KUKA KRL program: f1_Kuka_APT215T02S15.SRC

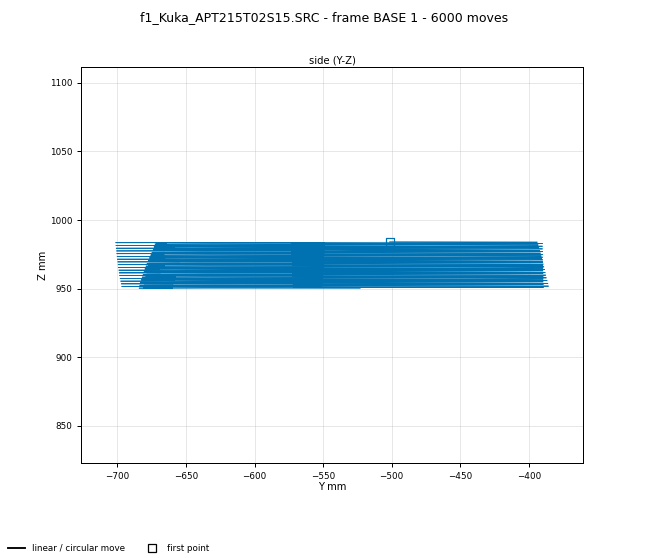
[picture p0: tool path of f1_Kuka_APT215T02S15.SRC in frame BASE 1, 6000 of 6001 moves have a stored position in this frame; points joined in program order, loops and branches not executed]
&ACCESS RVP
&REL 2
&PARAM TEMPLATE = C:\KRC\Roboter\Template\vorgabe
&PARAM EDITMASK = *
DEF f1_Kuka_APT215T02S15()


;FOLD INI;%{PE}%V3.2.0,%MKUKATPBASIS,%CINIT,%VCOMMON,%P
  ;FOLD BAS INI;%{E}%V3.2.0,%MKUKATPBASIS,%CINIT,%VINIT,%P
    GLOBAL INTERRUPT DECL 3 WHEN $STOPMESS==TRUE DO IR_STOPM ( )
    INTERRUPT ON 3
    BAS (#INITMOV,0 )
  ;ENDFOLD (BAS INI)
  ;FOLD USER INI;%{E}%V3.2.0,%MKUKATPUSER,%CINIT,%VINIT,%P
    ;Make your modifications here
  ;ENDFOLD (USER INI)
;ENDFOLD (INI)


;*** Make Null PTP Move
  PTP $pos_act

;*** Auto Load The Correct TOOL Data
  $tool=tool_data[2]

;*** Auto Load The Correct BASE Data
  $base=base_data[1]

  $ADVANCE = 5

;*** Restate Last Velocity
MMPM(30000.0)
SetRPM(8000)
LIN {X -0.285,Y -501.480,Z 984.115,A 0.000,B 0.000,C 90.000,E1 236.707} C_DIS
LIN {X 0.055,Y -498.844,Z 984.108,A 0.000,B 0.000,C 90.000,E1 235.468} C_DIS
LIN {X 0.071,Y -494.695,Z 984.098,A 0.000,B 0.000,C 90.000,E1 233.657} C_DIS
LIN {X -0.059,Y -492.503,Z 984.093,A 0.000,B 0.000,C 90.000,E1 232.763} C_DIS
LIN {X 0.019,Y -488.185,Z 984.083,A 0.000,B 0.000,C 90.000,E1 230.928} C_DIS
LIN {X 0.171,Y -484.612,Z 984.075,A 0.000,B 0.000,C 90.000,E1 229.380} C_DIS
LIN {X 0.130,Y -479.643,Z 984.063,A 0.000,B 0.000,C 90.000,E1 227.229} C_DIS
LIN {X -0.171,Y -475.684,Z 984.052,A 0.000,B 0.000,C 90.000,E1 225.405} C_DIS
LIN {X 0.017,Y -472.371,Z 984.044,A 0.000,B 0.000,C 90.000,E1 223.824} C_DIS
LIN {X 0.143,Y -468.887,Z 984.035,A 0.000,B 0.000,C 90.000,E1 222.243} C_DIS
LIN {X -0.119,Y -465.376,Z 984.026,A 0.000,B 0.000,C 90.000,E1 220.701} C_DIS
LIN {X 0.008,Y -461.153,Z 984.016,A 0.000,B 0.000,C 90.000,E1 218.785} C_DIS
LIN {X -0.234,Y -456.180,Z 984.003,A 0.000,B 0.000,C 90.000,E1 216.583} C_DIS
LIN {X 0.053,Y -453.348,Z 983.996,A 0.000,B 0.000,C 90.000,E1 215.264} C_DIS
LIN {X -0.282,Y -449.138,Z 983.985,A 0.000,B 0.000,C 90.000,E1 213.372} C_DIS
LIN {X -0.043,Y -445.627,Z 983.976,A 0.000,B 0.000,C 90.000,E1 211.720} C_DIS
LIN {X 0.037,Y -442.148,Z 983.967,A 0.000,B 0.000,C 90.000,E1 210.079} C_DIS
LIN {X 0.229,Y -439.200,Z 983.960,A 0.000,B 0.000,C 90.000,E1 208.743} C_DIS
LIN {X 0.220,Y -433.424,Z 983.945,A 0.000,B 0.000,C 90.000,E1 206.104} C_DIS
LIN {X -0.144,Y -430.325,Z 983.938,A 0.000,B 0.000,C 90.000,E1 204.823} C_DIS
LIN {X 0.213,Y -425.721,Z 983.927,A 0.000,B 0.000,C 90.000,E1 202.770} C_DIS
LIN {X 0.085,Y -420.612,Z 983.914,A 0.000,B 0.000,C 90.000,E1 200.429} C_DIS
LIN {X 0.213,Y -414.989,Z 983.898,A 0.000,B 0.000,C 90.000,E1 197.692} C_DIS
LIN {X 0.183,Y -409.982,Z 983.883,A 0.000,B 0.000,C 90.000,E1 194.954} C_DIS
LIN {X 0.056,Y -407.467,Z 983.876,A 0.000,B 0.000,C 90.000,E1 193.592} C_DIS
LIN {X -0.202,Y -405.003,Z 983.868,A 0.000,B 0.000,C 90.000,E1 192.243} C_DIS
LIN {X -0.103,Y -401.708,Z 983.858,A 0.000,B 0.000,C 90.000,E1 190.489} C_DIS
LIN {X -0.128,Y -399.174,Z 983.850,A 0.000,B 0.000,C 90.000,E1 189.095} C_DIS
LIN {X 0.168,Y -396.164,Z 983.841,A 0.000,B 0.000,C 90.000,E1 187.296} C_DIS
LIN {X 0.061,Y -395.147,Z 983.837,A 0.000,B 0.000,C 90.000,E1 186.606} C_DIS
LIN {X -0.088,Y -394.070,Z 983.831,A 0.000,B 0.000,C 90.000,E1 185.568} C_DIS
LIN {X -0.208,Y -393.751,Z 983.827,A 0.000,B 0.000,C 90.000,E1 184.878} C_DIS
LIN {X 0.062,Y -393.914,Z 983.823,A 0.000,B 0.000,C 90.000,E1 184.131} C_DIS
LIN {X -0.062,Y -394.851,Z 983.819,A 0.000,B 0.000,C 90.000,E1 183.440} C_DIS
LIN {X -0.092,Y -396.130,Z 983.816,A 0.000,B 0.000,C 90.000,E1 182.922} C_DIS
LIN {X -0.126,Y -399.219,Z 983.812,A 0.000,B 0.000,C 90.000,E1 182.178} C_DIS
LIN {X -0.178,Y -401.986,Z 983.809,A 0.000,B 0.000,C 90.000,E1 181.718} C_DIS
LIN {X -0.127,Y -405.589,Z 983.807,A 0.000,B 0.000,C 90.000,E1 181.203} C_DIS
LIN {X -0.089,Y -413.849,Z 983.802,A 0.000,B 0.000,C 90.000,E1 180.286} C_DIS
LIN {X -0.065,Y -430.114,Z 983.793,A 0.000,B 0.000,C 90.000,E1 178.682} C_DIS
LIN {X -0.102,Y -437.269,Z 983.789,A 0.000,B 0.000,C 90.000,E1 177.993} C_DIS
LIN {X -0.024,Y -444.519,Z 983.785,A 0.000,B 0.000,C 90.000,E1 177.249} C_DIS
LIN {X -0.047,Y -454.485,Z 983.779,A 0.000,B 0.000,C 90.000,E1 176.216} C_DIS
LIN {X -0.161,Y -462.529,Z 983.774,A 0.000,B 0.000,C 90.000,E1 175.355} C_DIS
LIN {X -0.135,Y -470.477,Z 983.769,A 0.000,B 0.000,C 90.000,E1 174.432} C_DIS
LIN {X 0.088,Y -477.048,Z 983.765,A 0.000,B 0.000,C 90.000,E1 173.628} C_DIS
LIN {X -0.152,Y -481.893,Z 983.761,A 0.000,B 0.000,C 90.000,E1 173.053} C_DIS
LIN {X -0.064,Y -492.291,Z 983.754,A 0.000,B 0.000,C 90.000,E1 171.659} C_DIS
LIN {X 0.053,Y -499.067,Z 983.749,A 0.000,B 0.000,C 90.000,E1 170.735} C_DIS
LIN {X -0.052,Y -508.367,Z 983.741,A 0.000,B 0.000,C 90.000,E1 169.398} C_DIS
LIN {X 0.115,Y -515.180,Z 983.735,A 0.000,B 0.000,C 90.000,E1 168.342} C_DIS
LIN {X 0.075,Y -524.600,Z 983.727,A 0.000,B 0.000,C 90.000,E1 166.881} C_DIS
LIN {X -0.025,Y -532.594,Z 983.720,A 0.000,B 0.000,C 90.000,E1 165.589} C_DIS
LIN {X 0.135,Y -540.298,Z 983.713,A 0.000,B 0.000,C 90.000,E1 164.283} C_DIS
LIN {X 0.199,Y -546.883,Z 983.706,A 0.000,B 0.000,C 90.000,E1 163.142} C_DIS
LIN {X -0.163,Y -553.385,Z 983.700,A 0.000,B 0.000,C 90.000,E1 162.054} C_DIS
LIN {X -0.012,Y -562.621,Z 983.691,A 0.000,B 0.000,C 90.000,E1 160.369} C_DIS
LIN {X -0.098,Y -565.614,Z 983.688,A 0.000,B 0.000,C 90.000,E1 159.826} C_DIS
LIN {X 0.079,Y -570.773,Z 983.683,A 0.000,B 0.000,C 90.000,E1 158.847} C_DIS
LIN {X 0.154,Y -576.864,Z 983.676,A 0.000,B 0.000,C 90.000,E1 157.614} C_DIS
LIN {X 0.021,Y -582.436,Z 983.669,A 0.000,B 0.000,C 90.000,E1 156.410} C_DIS
LIN {X -0.013,Y -585.413,Z 983.665,A 0.000,B 0.000,C 90.000,E1 155.741} C_DIS
LIN {X 0.152,Y -588.856,Z 983.661,A 0.000,B 0.000,C 90.000,E1 154.921} C_DIS
LIN {X -0.073,Y -590.996,Z 983.658,A 0.000,B 0.000,C 90.000,E1 154.409} C_DIS
LIN {X 0.148,Y -593.860,Z 983.653,A 0.000,B 0.000,C 90.000,E1 153.589} C_DIS
LIN {X 0.053,Y -597.438,Z 983.648,A 0.000,B 0.000,C 90.000,E1 152.538} C_DIS
LIN {X -0.344,Y -601.601,Z 983.640,A 0.000,B 0.000,C 90.000,E1 151.257} C_DIS
LIN {X -0.216,Y -607.066,Z 983.630,A 0.000,B 0.000,C 90.000,E1 149.410} C_DIS
LIN {X -0.160,Y -612.486,Z 983.620,A 0.000,B 0.000,C 90.000,E1 147.582} C_DIS
LIN {X -0.183,Y -618.603,Z 983.608,A 0.000,B 0.000,C 90.000,E1 145.515} C_DIS
LIN {X -0.352,Y -623.180,Z 983.600,A 0.000,B 0.000,C 90.000,E1 143.989} C_DIS
LIN {X -0.225,Y -628.419,Z 983.590,A 0.000,B 0.000,C 90.000,E1 142.190} C_DIS
LIN {X 0.179,Y -632.139,Z 983.583,A 0.000,B 0.000,C 90.000,E1 140.884} C_DIS
LIN {X 0.151,Y -635.816,Z 983.576,A 0.000,B 0.000,C 90.000,E1 139.622} C_DIS
LIN {X -0.012,Y -640.782,Z 983.566,A 0.000,B 0.000,C 90.000,E1 137.877} C_DIS
LIN {X -0.102,Y -645.956,Z 983.556,A 0.000,B 0.000,C 90.000,E1 136.134} C_DIS
LIN {X 0.340,Y -652.259,Z 983.545,A 0.000,B 0.000,C 90.000,E1 134.109} C_DIS
LIN {X 0.024,Y -659.797,Z 983.533,A 0.000,B 0.000,C 90.000,E1 131.919} C_DIS
LIN {X -0.052,Y -665.162,Z 983.525,A 0.000,B 0.000,C 90.000,E1 130.458} C_DIS
LIN {X -0.036,Y -669.484,Z 983.518,A 0.000,B 0.000,C 90.000,E1 129.241} C_DIS
LIN {X -0.271,Y -674.290,Z 983.510,A 0.000,B 0.000,C 90.000,E1 127.810} C_DIS
LIN {X -0.005,Y -677.255,Z 983.505,A 0.000,B 0.000,C 90.000,E1 126.824} C_DIS
LIN {X 0.315,Y -680.816,Z 983.498,A 0.000,B 0.000,C 90.000,E1 125.598} C_DIS
LIN {X -0.279,Y -683.674,Z 983.493,A 0.000,B 0.000,C 90.000,E1 124.692} C_DIS
LIN {X 0.110,Y -686.255,Z 983.487,A 0.000,B 0.000,C 90.000,E1 123.706} C_DIS
LIN {X -0.218,Y -689.353,Z 983.481,A 0.000,B 0.000,C 90.000,E1 122.546} C_DIS
LIN {X -0.141,Y -691.866,Z 983.476,A 0.000,B 0.000,C 90.000,E1 121.592} C_DIS
LIN {X -0.036,Y -693.620,Z 983.472,A 0.000,B 0.000,C 90.000,E1 120.875} C_DIS
LIN {X 0.089,Y -695.708,Z 983.466,A 0.000,B 0.000,C 90.000,E1 119.922} C_DIS
LIN {X -0.015,Y -696.670,Z 983.464,A 0.000,B 0.000,C 90.000,E1 119.461} C_DIS
LIN {X 0.143,Y -697.815,Z 983.460,A 0.000,B 0.000,C 90.000,E1 118.743} C_DIS
LIN {X 0.313,Y -698.687,Z 983.456,A 0.000,B 0.000,C 90.000,E1 118.025} C_DIS
LIN {X -0.185,Y -699.537,Z 983.451,A 0.000,B 0.000,C 90.000,E1 117.129} C_DIS
LIN {X 0.232,Y -700.567,Z 983.444,A 0.000,B 0.000,C 90.000,E1 115.924} C_DIS
LIN {X 0.421,Y -701.035,Z 983.440,A 0.000,B 0.000,C 90.000,E1 115.207} C_DIS
LIN {X 0.309,Y -701.247,Z 983.436,A 0.000,B 0.000,C 90.000,E1 114.515} C_DIS
LIN {X -0.346,Y -701.281,Z 983.435,A 0.000,B 0.000,C 90.000,E1 114.335} C_DIS
LIN {X 0.199,Y -700.940,Z 983.432,A 0.000,B 0.000,C 90.000,E1 113.823} C_DIS
LIN {X 0.189,Y -700.708,Z 983.431,A 0.000,B 0.000,C 90.000,E1 113.590} C_DIS
LIN {X 0.085,Y -699.116,Z 983.429,A 0.000,B 0.000,C 90.000,E1 113.131} C_DIS
LIN {X 0.075,Y -698.093,Z 983.427,A 0.000,B 0.000,C 90.000,E1 112.898} C_DIS
LIN {X 0.206,Y -697.243,Z 983.427,A 0.000,B 0.000,C 90.000,E1 112.770} C_DIS
LIN {X -0.161,Y -692.450,Z 983.424,A 0.000,B 0.000,C 90.000,E1 112.333} C_DIS
LIN {X -0.010,Y -690.903,Z 983.423,A 0.000,B 0.000,C 90.000,E1 112.206} C_DIS
LIN {X 0.296,Y -688.613,Z 983.423,A 0.000,B 0.000,C 90.000,E1 112.078} C_DIS
LIN {X -0.293,Y -685.802,Z 983.422,A 0.000,B 0.000,C 90.000,E1 112.025} C_DIS
LIN {X -0.134,Y -683.818,Z 983.422,A 0.000,B 0.000,C 90.000,E1 111.950} C_DIS
LIN {X 0.163,Y -676.154,Z 983.421,A 0.000,B 0.000,C 90.000,E1 111.770} C_DIS
LIN {X -0.011,Y -675.079,Z 983.421,A 0.000,B 0.000,C 90.000,E1 111.770} C_DIS
LIN {X -0.136,Y -670.289,Z 983.421,A 0.000,B 0.000,C 90.000,E1 111.770} C_DIS
LIN {X -0.175,Y -623.351,Z 983.421,A 0.000,B 0.000,C 90.000,E1 111.770} C_DIS
LIN {X 0.338,Y -616.816,Z 983.420,A 0.000,B 0.000,C 90.000,E1 111.589} C_DIS
LIN {X 0.089,Y -609.967,Z 983.419,A 0.000,B 0.000,C 90.000,E1 111.408} C_DIS
LIN {X -0.162,Y -603.110,Z 983.417,A 0.000,B 0.000,C 90.000,E1 111.153} C_DIS
LIN {X 0.051,Y -596.699,Z 983.416,A 0.000,B 0.000,C 90.000,E1 110.791} C_DIS
LIN {X 0.283,Y -589.920,Z 983.413,A 0.000,B 0.000,C 90.000,E1 110.301} C_DIS
LIN {X 0.083,Y -578.734,Z 983.408,A 0.000,B 0.000,C 90.000,E1 109.450} C_DIS
LIN {X -0.200,Y -574.341,Z 983.406,A 0.000,B 0.000,C 90.000,E1 109.141} C_DIS
LIN {X 0.100,Y -566.102,Z 983.403,A 0.000,B 0.000,C 90.000,E1 108.598} C_DIS
LIN {X -0.139,Y -551.469,Z 983.399,A 0.000,B 0.000,C 90.000,E1 107.873} C_DIS
LIN {X -0.110,Y -549.548,Z 983.398,A 0.000,B 0.000,C 90.000,E1 107.692} C_DIS
LIN {X -0.148,Y -549.526,Z 983.398,A 0.000,B 0.000,C 90.000,E1 107.692} C_DIS
LIN {X 0.154,Y -549.085,Z 983.397,A 0.000,B 0.000,C 90.000,E1 107.402} C_DIS
LIN {X -0.064,Y -549.295,Z 983.391,A 0.000,B 0.000,C 90.000,E1 106.441} C_DIS
LIN {X 0.104,Y -549.806,Z 983.385,A 0.000,B 0.000,C 90.000,E1 105.300} C_DIS
LIN {X -0.050,Y -551.809,Z 983.366,A 0.000,B 0.000,C 90.000,E1 101.951} C_DIS
LIN {X -0.177,Y -553.911,Z 983.354,A 0.000,B 0.000,C 90.000,E1 99.726} C_DIS
LIN {X -0.277,Y -555.403,Z 983.346,A 0.000,B 0.000,C 90.000,E1 98.341} C_DIS
LIN {X 0.283,Y -556.801,Z 983.339,A 0.000,B 0.000,C 90.000,E1 96.891} C_DIS
LIN {X 0.110,Y -557.762,Z 983.332,A 0.000,B 0.000,C 90.000,E1 95.796} C_DIS
LIN {X 0.025,Y -558.746,Z 983.325,A 0.000,B 0.000,C 90.000,E1 94.416} C_DIS
LIN {X -0.046,Y -559.600,Z 983.317,A 0.000,B 0.000,C 90.000,E1 93.037} C_DIS
LIN {X -0.139,Y -560.331,Z 983.309,A 0.000,B 0.000,C 90.000,E1 91.661} C_DIS
LIN {X 0.235,Y -560.916,Z 983.303,A 0.000,B 0.000,C 90.000,E1 90.516} C_DIS
LIN {X 0.158,Y -561.493,Z 983.295,A 0.000,B 0.000,C 90.000,E1 89.141} C_DIS
LIN {X 0.103,Y -561.843,Z 983.288,A 0.000,B 0.000,C 90.000,E1 87.764} C_DIS
LIN {X 0.149,Y -562.155,Z 983.279,A 0.000,B 0.000,C 90.000,E1 86.102} C_DIS
LIN {X 0.278,Y -562.386,Z 983.269,A 0.000,B 0.000,C 90.000,E1 84.432} C_DIS
LIN {X -0.060,Y -562.664,Z 983.259,A 0.000,B 0.000,C 90.000,E1 82.534} C_DIS
LIN {X -0.257,Y -563.167,Z 983.248,A 0.000,B 0.000,C 90.000,E1 80.622} C_DIS
LIN {X -0.186,Y -564.058,Z 983.236,A 0.000,B 0.000,C 90.000,E1 78.409} C_DIS
LIN {X 0.205,Y -564.787,Z 983.228,A 0.000,B 0.000,C 90.000,E1 76.992} C_DIS
LIN {X 0.024,Y -566.192,Z 983.216,A 0.000,B 0.000,C 90.000,E1 74.810} C_DIS
LIN {X -0.152,Y -567.537,Z 983.205,A 0.000,B 0.000,C 90.000,E1 72.906} C_DIS
LIN {X 0.088,Y -568.474,Z 983.197,A 0.000,B 0.000,C 90.000,E1 71.511} C_DIS
LIN {X 0.007,Y -569.194,Z 983.191,A 0.000,B 0.000,C 90.000,E1 70.423} C_DIS
LIN {X -0.257,Y -569.933,Z 983.184,A 0.000,B 0.000,C 90.000,E1 69.082} C_DIS
LIN {X -0.126,Y -570.537,Z 983.178,A 0.000,B 0.000,C 90.000,E1 67.975} C_DIS
LIN {X 0.186,Y -571.178,Z 983.169,A 0.000,B 0.000,C 90.000,E1 66.305} C_DIS
LIN {X 0.215,Y -571.766,Z 983.159,A 0.000,B 0.000,C 90.000,E1 64.665} C_DIS
LIN {X -0.005,Y -572.187,Z 983.150,A 0.000,B 0.000,C 90.000,E1 63.050} C_DIS
LIN {X -0.207,Y -572.573,Z 983.141,A 0.000,B 0.000,C 90.000,E1 61.435} C_DIS
LIN {X 0.034,Y -572.753,Z 983.134,A 0.000,B 0.000,C 90.000,E1 60.049} C_DIS
LIN {X 0.149,Y -572.883,Z 983.128,A 0.000,B 0.000,C 90.000,E1 58.948} C_DIS
LIN {X 0.062,Y -573.095,Z 983.122,A 0.000,B 0.000,C 90.000,E1 57.867} C_DIS
LIN {X 0.113,Y -573.180,Z 983.114,A 0.000,B 0.000,C 90.000,E1 56.501} C_DIS
LIN {X -0.311,Y -573.190,Z 983.106,A 0.000,B 0.000,C 90.000,E1 55.182} C_DIS
LIN {X -0.079,Y -573.027,Z 983.100,A 0.000,B 0.000,C 90.000,E1 54.069} C_DIS
LIN {X -0.040,Y -572.406,Z 983.091,A 0.000,B 0.000,C 90.000,E1 52.431} C_DIS
LIN {X 0.059,Y -571.777,Z 983.085,A 0.000,B 0.000,C 90.000,E1 51.331} C_DIS
LIN {X -0.290,Y -570.953,Z 983.079,A 0.000,B 0.000,C 90.000,E1 50.275} C_DIS
LIN {X -0.337,Y -570.222,Z 983.075,A 0.000,B 0.000,C 90.000,E1 49.461} C_DIS
LIN {X -0.021,Y -569.358,Z 983.070,A 0.000,B 0.000,C 90.000,E1 48.609} C_DIS
LIN {X -0.092,Y -568.313,Z 983.066,A 0.000,B 0.000,C 90.000,E1 47.796} C_DIS
LIN {X -0.215,Y -567.076,Z 983.061,A 0.000,B 0.000,C 90.000,E1 46.986} C_DIS
LIN {X 0.067,Y -565.666,Z 983.056,A 0.000,B 0.000,C 90.000,E1 46.134} C_DIS
LIN {X 0.238,Y -564.660,Z 983.053,A 0.000,B 0.000,C 90.000,E1 45.567} C_DIS
LIN {X -0.234,Y -562.296,Z 983.047,A 0.000,B 0.000,C 90.000,E1 44.514} C_DIS
LIN {X -0.085,Y -560.979,Z 983.044,A 0.000,B 0.000,C 90.000,E1 43.947} C_DIS
LIN {X 0.128,Y -558.736,Z 983.040,A 0.000,B 0.000,C 90.000,E1 43.095} C_DIS
LIN {X 0.248,Y -557.113,Z 983.036,A 0.000,B 0.000,C 90.000,E1 42.528} C_DIS
LIN {X -0.020,Y -555.357,Z 983.033,A 0.000,B 0.000,C 90.000,E1 42.000} C_DIS
LIN {X 0.132,Y -552.392,Z 983.029,A 0.000,B 0.000,C 90.000,E1 41.148} C_DIS
LIN {X -0.108,Y -549.061,Z 983.024,A 0.000,B 0.000,C 90.000,E1 40.334} C_DIS
LIN {X 0.146,Y -547.298,Z 983.022,A 0.000,B 0.000,C 90.000,E1 39.886} C_DIS
LIN {X 0.008,Y -544.117,Z 983.018,A 0.000,B 0.000,C 90.000,E1 39.197} C_DIS
LIN {X 0.257,Y -540.697,Z 983.014,A 0.000,B 0.000,C 90.000,E1 38.463} C_DIS
LIN {X -0.270,Y -535.557,Z 983.008,A 0.000,B 0.000,C 90.000,E1 37.523} C_DIS
LIN {X -0.265,Y -530.880,Z 983.004,A 0.000,B 0.000,C 90.000,E1 36.664} C_DIS
LIN {X -0.312,Y -525.968,Z 982.999,A 0.000,B 0.000,C 90.000,E1 35.804} C_DIS
LIN {X 0.136,Y -519.801,Z 982.993,A 0.000,B 0.000,C 90.000,E1 34.739} C_DIS
LIN {X -0.154,Y -514.968,Z 982.989,A 0.000,B 0.000,C 90.000,E1 34.040} C_DIS
LIN {X 0.020,Y -512.025,Z 982.987,A 0.000,B 0.000,C 90.000,E1 33.579} C_DIS
LIN {X 0.089,Y -506.642,Z 982.982,A 0.000,B 0.000,C 90.000,E1 32.832} C_DIS
LIN {X -0.203,Y -503.270,Z 982.980,A 0.000,B 0.000,C 90.000,E1 32.418} C_DIS
LIN {X -0.018,Y -498.482,Z 982.977,A 0.000,B 0.000,C 90.000,E1 31.799} C_DIS
LIN {X -0.127,Y -493.269,Z 982.973,A 0.000,B 0.000,C 90.000,E1 31.209} C_DIS
LIN {X 0.126,Y -487.817,Z 982.970,A 0.000,B 0.000,C 90.000,E1 30.590} C_DIS
LIN {X 0.255,Y -482.201,Z 982.967,A 0.000,B 0.000,C 90.000,E1 30.001} C_DIS
LIN {X -0.086,Y -473.618,Z 982.962,A 0.000,B 0.000,C 90.000,E1 29.205} C_DIS
LIN {X 0.083,Y -464.827,Z 982.958,A 0.000,B 0.000,C 90.000,E1 28.359} C_DIS
LIN {X -0.213,Y -455.844,Z 982.953,A 0.000,B 0.000,C 90.000,E1 27.590} C_DIS
LIN {X 0.208,Y -445.140,Z 982.948,A 0.000,B 0.000,C 90.000,E1 26.616} C_DIS
LIN {X 0.191,Y -424.073,Z 982.938,A 0.000,B 0.000,C 90.000,E1 24.771} C_DIS
LIN {X 0.075,Y -410.898,Z 982.931,A 0.000,B 0.000,C 90.000,E1 23.515} C_DIS
LIN {X 0.048,Y -400.755,Z 982.925,A 0.000,B 0.000,C 90.000,E1 22.461} C_DIS
LIN {X -0.235,Y -395.452,Z 982.921,A 0.000,B 0.000,C 90.000,E1 21.844} C_DIS
LIN {X 0.045,Y -393.670,Z 982.920,A 0.000,B 0.000,C 90.000,E1 21.535} C_DIS
LIN {X 0.058,Y -392.004,Z 982.918,A 0.000,B 0.000,C 90.000,E1 21.227} C_DIS
LIN {X 0.123,Y -391.011,Z 982.916,A 0.000,B 0.000,C 90.000,E1 20.918} C_DIS
LIN {X -0.110,Y -390.077,Z 982.913,A 0.000,B 0.000,C 90.000,E1 20.301} C_DIS
LIN {X -0.027,Y -389.979,Z 982.909,A 0.000,B 0.000,C 90.000,E1 19.577} C_DIS
LIN {X -0.058,Y -393.201,Z 982.889,A 0.000,B 0.000,C 90.000,E1 16.024} C_DIS
LIN {X 0.001,Y -395.272,Z 982.879,A 0.000,B 0.000,C 90.000,E1 14.245} C_DIS
LIN {X 0.064,Y -398.050,Z 982.867,A 0.000,B 0.000,C 90.000,E1 12.119} C_DIS
LIN {X -0.001,Y -403.044,Z 982.850,A 0.000,B 0.000,C 90.000,E1 8.973} C_DIS
LIN {X -0.076,Y -408.132,Z 982.834,A 0.000,B 0.000,C 90.000,E1 6.201} C_DIS
LIN {X -0.036,Y -414.656,Z 982.817,A 0.000,B 0.000,C 90.000,E1 3.094} C_DIS
LIN {X 0.042,Y -418.443,Z 982.808,A 0.000,B 0.000,C 90.000,E1 1.375} C_DIS
LIN {X 0.093,Y -420.374,Z 982.804,A 0.000,B 0.000,C 90.000,E1 0.688} C_DIS
LIN {X -0.182,Y -422.321,Z 982.801,A 0.000,B 0.000,C 90.000,E1 0.229} C_DIS
LIN {X 0.000,Y -423.349,Z 982.800,A 0.000,B 0.000,C 90.000,E1 360.000} C_DIS
LIN {X 0.161,Y -424.635,Z 982.799,A 0.000,B 0.000,C 90.000,E1 359.771} C_DIS
LIN {X -0.139,Y -427.560,Z 982.797,A 0.000,B 0.000,C 90.000,E1 359.427} C_DIS
LIN {X -0.113,Y -429.052,Z 982.796,A 0.000,B 0.000,C 90.000,E1 359.255} C_DIS
LIN {X -0.106,Y -434.383,Z 982.794,A 0.000,B 0.000,C 90.000,E1 358.854} C_DIS
LIN {X -0.209,Y -447.063,Z 982.790,A 0.000,B 0.000,C 90.000,E1 358.165} C_DIS
LIN {X -0.226,Y -460.540,Z 982.786,A 0.000,B 0.000,C 90.000,E1 357.421} C_DIS
LIN {X -0.107,Y -470.730,Z 982.782,A 0.000,B 0.000,C 90.000,E1 356.846} C_DIS
LIN {X 0.101,Y -485.521,Z 982.778,A 0.000,B 0.000,C 90.000,E1 355.988} C_DIS
LIN {X 0.195,Y -495.296,Z 982.775,A 0.000,B 0.000,C 90.000,E1 355.412} C_DIS
LIN {X -0.137,Y -506.369,Z 982.771,A 0.000,B 0.000,C 90.000,E1 354.780} C_DIS
LIN {X -0.006,Y -514.242,Z 982.768,A 0.000,B 0.000,C 90.000,E1 354.261} C_DIS
LIN {X -0.094,Y -521.992,Z 982.765,A 0.000,B 0.000,C 90.000,E1 353.742} C_DIS
LIN {X 0.120,Y -526.435,Z 982.763,A 0.000,B 0.000,C 90.000,E1 353.394} C_DIS
LIN {X -0.093,Y -532.000,Z 982.761,A 0.000,B 0.000,C 90.000,E1 352.996} C_DIS
LIN {X -0.166,Y -539.135,Z 982.758,A 0.000,B 0.000,C 90.000,E1 352.413} C_DIS
LIN {X -0.219,Y -544.309,Z 982.755,A 0.000,B 0.000,C 90.000,E1 351.951} C_DIS
LIN {X 0.305,Y -550.808,Z 982.752,A 0.000,B 0.000,C 90.000,E1 351.254} C_DIS
LIN {X 0.115,Y -555.841,Z 982.749,A 0.000,B 0.000,C 90.000,E1 350.735} C_DIS
LIN {X -0.142,Y -560.539,Z 982.746,A 0.000,B 0.000,C 90.000,E1 350.208} C_DIS
LIN {X -0.087,Y -565.859,Z 982.742,A 0.000,B 0.000,C 90.000,E1 349.511} C_DIS
LIN {X 0.259,Y -569.810,Z 982.739,A 0.000,B 0.000,C 90.000,E1 348.926} C_DIS
LIN {X -0.165,Y -574.246,Z 982.735,A 0.000,B 0.000,C 90.000,E1 348.285} C_DIS
LIN {X 0.242,Y -577.552,Z 982.732,A 0.000,B 0.000,C 90.000,E1 347.701} C_DIS
LIN {X -0.102,Y -584.341,Z 982.725,A 0.000,B 0.000,C 90.000,E1 346.520} C_DIS
LIN {X -0.190,Y -587.182,Z 982.722,A 0.000,B 0.000,C 90.000,E1 345.992} C_DIS
LIN {X -0.128,Y -594.507,Z 982.714,A 0.000,B 0.000,C 90.000,E1 344.519} C_DIS
LIN {X -0.354,Y -601.240,Z 982.706,A 0.000,B 0.000,C 90.000,E1 343.087} C_DIS
LIN {X -0.168,Y -603.552,Z 982.703,A 0.000,B 0.000,C 90.000,E1 342.543} C_DIS
LIN {X -0.017,Y -609.021,Z 982.696,A 0.000,B 0.000,C 90.000,E1 341.221} C_DIS
LIN {X 0.162,Y -612.119,Z 982.691,A 0.000,B 0.000,C 90.000,E1 340.423} C_DIS
LIN {X 0.127,Y -615.971,Z 982.686,A 0.000,B 0.000,C 90.000,E1 339.390} C_DIS
LIN {X 0.114,Y -620.326,Z 982.678,A 0.000,B 0.000,C 90.000,E1 338.103} C_DIS
LIN {X -0.167,Y -624.410,Z 982.671,A 0.000,B 0.000,C 90.000,E1 336.847} C_DIS
LIN {X 0.200,Y -628.137,Z 982.664,A 0.000,B 0.000,C 90.000,E1 335.537} C_DIS
LIN {X 0.023,Y -630.916,Z 982.659,A 0.000,B 0.000,C 90.000,E1 334.537} C_DIS
LIN {X 0.151,Y -633.401,Z 982.653,A 0.000,B 0.000,C 90.000,E1 333.512} C_DIS
LIN {X 0.314,Y -635.720,Z 982.647,A 0.000,B 0.000,C 90.000,E1 332.487} C_DIS
LIN {X 0.043,Y -638.867,Z 982.639,A 0.000,B 0.000,C 90.000,E1 331.001} C_DIS
LIN {X 0.078,Y -641.270,Z 982.632,A 0.000,B 0.000,C 90.000,E1 329.744} C_DIS
LIN {X 0.031,Y -642.634,Z 982.628,A 0.000,B 0.000,C 90.000,E1 328.997} C_DIS
LIN {X 0.125,Y -644.591,Z 982.621,A 0.000,B 0.000,C 90.000,E1 327.740} C_DIS
LIN {X -0.016,Y -645.946,Z 982.615,A 0.000,B 0.000,C 90.000,E1 326.755} C_DIS
LIN {X 0.047,Y -647.193,Z 982.610,A 0.000,B 0.000,C 90.000,E1 325.754} C_DIS
LIN {X -0.150,Y -648.376,Z 982.603,A 0.000,B 0.000,C 90.000,E1 324.529} C_DIS
LIN {X -0.261,Y -649.439,Z 982.595,A 0.000,B 0.000,C 90.000,E1 323.050} C_DIS
LIN {X 0.030,Y -650.185,Z 982.586,A 0.000,B 0.000,C 90.000,E1 321.537} C_DIS
LIN {X 0.300,Y -650.750,Z 982.580,A 0.000,B 0.000,C 90.000,E1 320.275} C_DIS
LIN {X 0.034,Y -651.497,Z 982.570,A 0.000,B 0.000,C 90.000,E1 318.566} C_DIS
LIN {X 0.122,Y -652.867,Z 982.559,A 0.000,B 0.000,C 90.000,E1 316.581} C_DIS
LIN {X 0.298,Y -654.128,Z 982.549,A 0.000,B 0.000,C 90.000,E1 314.838} C_DIS
LIN {X 0.430,Y -655.871,Z 982.537,A 0.000,B 0.000,C 90.000,E1 312.609} C_DIS
LIN {X -0.122,Y -656.439,Z 982.533,A 0.000,B 0.000,C 90.000,E1 311.919} C_DIS
LIN {X -0.247,Y -657.334,Z 982.526,A 0.000,B 0.000,C 90.000,E1 310.701} C_DIS
LIN {X 0.145,Y -658.062,Z 982.519,A 0.000,B 0.000,C 90.000,E1 309.439} C_DIS
LIN {X 0.078,Y -658.567,Z 982.514,A 0.000,B 0.000,C 90.000,E1 308.463} C_DIS
LIN {X 0.078,Y -659.144,Z 982.507,A 0.000,B 0.000,C 90.000,E1 307.237} C_DIS
LIN {X 0.056,Y -659.433,Z 982.503,A 0.000,B 0.000,C 90.000,E1 306.503} C_DIS
LIN {X 0.183,Y -659.756,Z 982.492,A 0.000,B 0.000,C 90.000,E1 304.532} C_DIS
LIN {X 0.200,Y -660.834,Z 982.476,A 0.000,B 0.000,C 90.000,E1 301.592} C_DIS
LIN {X -0.199,Y -664.615,Z 982.454,A 0.000,B 0.000,C 90.000,E1 297.719} C_DIS
LIN {X -0.323,Y -668.087,Z 982.442,A 0.000,B 0.000,C 90.000,E1 295.540} C_DIS
LIN {X -0.412,Y -670.135,Z 982.435,A 0.000,B 0.000,C 90.000,E1 294.335} C_DIS
LIN {X -0.027,Y -671.593,Z 982.430,A 0.000,B 0.000,C 90.000,E1 293.334} C_DIS
LIN {X 0.303,Y -672.203,Z 982.427,A 0.000,B 0.000,C 90.000,E1 292.823} C_DIS
LIN {X -0.246,Y -672.657,Z 982.424,A 0.000,B 0.000,C 90.000,E1 292.386} C_DIS
LIN {X -0.170,Y -672.593,Z 982.422,A 0.000,B 0.000,C 90.000,E1 291.897} C_DIS
LIN {X -0.007,Y -672.413,Z 982.420,A 0.000,B 0.000,C 90.000,E1 291.642} C_DIS
LIN {X -0.092,Y -672.021,Z 982.419,A 0.000,B 0.000,C 90.000,E1 291.408} C_DIS
LIN {X 0.069,Y -671.483,Z 982.418,A 0.000,B 0.000,C 90.000,E1 291.153} C_DIS
LIN {X -0.014,Y -670.584,Z 982.416,A 0.000,B 0.000,C 90.000,E1 290.918} C_DIS
LIN {X -0.020,Y -667.906,Z 982.414,A 0.000,B 0.000,C 90.000,E1 290.556} C_DIS
LIN {X 0.124,Y -665.611,Z 982.413,A 0.000,B 0.000,C 90.000,E1 290.301} C_DIS
LIN {X 0.193,Y -664.113,Z 982.412,A 0.000,B 0.000,C 90.000,E1 290.174} C_DIS
LIN {X 0.190,Y -658.008,Z 982.410,A 0.000,B 0.000,C 90.000,E1 289.758} C_DIS
LIN {X -0.161,Y -653.119,Z 982.408,A 0.000,B 0.000,C 90.000,E1 289.504} C_DIS
LIN {X 0.110,Y -648.358,Z 982.406,A 0.000,B 0.000,C 90.000,E1 289.141} C_DIS
LIN {X 0.072,Y -648.316,Z 982.406,A 0.000,B 0.000,C 90.000,E1 289.141} C_DIS
LIN {X -0.274,Y -648.212,Z 982.406,A 0.000,B 0.000,C 90.000,E1 289.141} C_DIS
LIN {X 0.301,Y -648.219,Z 982.406,A 0.000,B 0.000,C 90.000,E1 289.087} C_DIS
LIN {X -0.229,Y -648.971,Z 982.405,A 0.000,B 0.000,C 90.000,E1 288.852} C_DIS
LIN {X -0.165,Y -650.078,Z 982.403,A 0.000,B 0.000,C 90.000,E1 288.598} C_DIS
LIN {X -0.273,Y -652.041,Z 982.401,A 0.000,B 0.000,C 90.000,E1 288.236} C_DIS
LIN {X 0.127,Y -655.993,Z 982.398,A 0.000,B 0.000,C 90.000,E1 287.583} C_DIS
LIN {X 0.024,Y -660.870,Z 982.393,A 0.000,B 0.000,C 90.000,E1 286.732} C_DIS
LIN {X -0.132,Y -663.954,Z 982.390,A 0.000,B 0.000,C 90.000,E1 286.134} C_DIS
LIN {X -0.313,Y -665.866,Z 982.387,A 0.000,B 0.000,C 90.000,E1 285.662} C_DIS
LIN {X 0.163,Y -667.422,Z 982.384,A 0.000,B 0.000,C 90.000,E1 285.134} C_DIS
LIN {X 0.085,Y -668.153,Z 982.383,A 0.000,B 0.000,C 90.000,E1 284.898} C_DIS
LIN {X 0.029,Y -669.720,Z 982.379,A 0.000,B 0.000,C 90.000,E1 284.175} C_DIS
LIN {X -0.182,Y -670.779,Z 982.375,A 0.000,B 0.000,C 90.000,E1 283.467} C_DIS
LIN {X 0.184,Y -671.330,Z 982.372,A 0.000,B 0.000,C 90.000,E1 282.952} C_DIS
LIN {X 0.057,Y -671.675,Z 982.369,A 0.000,B 0.000,C 90.000,E1 282.479} C_DIS
LIN {X -0.070,Y -671.855,Z 982.367,A 0.000,B 0.000,C 90.000,E1 282.007} C_DIS
LIN {X -0.266,Y -671.652,Z 982.363,A 0.000,B 0.000,C 90.000,E1 281.299} C_DIS
LIN {X 0.131,Y -671.369,Z 982.360,A 0.000,B 0.000,C 90.000,E1 280.782} C_DIS
LIN {X -0.006,Y -670.835,Z 982.357,A 0.000,B 0.000,C 90.000,E1 280.310} C_DIS
LIN {X -0.265,Y -670.093,Z 982.355,A 0.000,B 0.000,C 90.000,E1 279.849} C_DIS
LIN {X 0.243,Y -669.066,Z 982.352,A 0.000,B 0.000,C 90.000,E1 279.321} C_DIS
LIN {X -0.024,Y -667.684,Z 982.349,A 0.000,B 0.000,C 90.000,E1 278.859} C_DIS
LIN {X -0.109,Y -666.931,Z 982.348,A 0.000,B 0.000,C 90.000,E1 278.624} C_DIS
LIN {X 0.272,Y -665.147,Z 982.345,A 0.000,B 0.000,C 90.000,E1 278.106} C_DIS
LIN {X -0.014,Y -663.124,Z 982.343,A 0.000,B 0.000,C 90.000,E1 277.644} C_DIS
LIN {X 0.245,Y -659.902,Z 982.339,A 0.000,B 0.000,C 90.000,E1 277.011} C_DIS
LIN {X -0.100,Y -655.996,Z 982.336,A 0.000,B 0.000,C 90.000,E1 276.429} C_DIS
LIN {X 0.204,Y -652.390,Z 982.333,A 0.000,B 0.000,C 90.000,E1 275.910} C_DIS
LIN {X -0.165,Y -648.368,Z 982.330,A 0.000,B 0.000,C 90.000,E1 275.448} C_DIS
LIN {X -0.089,Y -642.787,Z 982.327,A 0.000,B 0.000,C 90.000,E1 274.821} C_DIS
LIN {X 0.158,Y -637.935,Z 982.324,A 0.000,B 0.000,C 90.000,E1 274.302} C_DIS
LIN {X 0.208,Y -631.774,Z 982.321,A 0.000,B 0.000,C 90.000,E1 273.726} C_DIS
LIN {X 0.268,Y -625.014,Z 982.318,A 0.000,B 0.000,C 90.000,E1 273.154} C_DIS
LIN {X 0.032,Y -617.651,Z 982.315,A 0.000,B 0.000,C 90.000,E1 272.636} C_DIS
LIN {X -0.061,Y -611.592,Z 982.312,A 0.000,B 0.000,C 90.000,E1 272.236} C_DIS
LIN {X 0.138,Y -604.992,Z 982.310,A 0.000,B 0.000,C 90.000,E1 271.835} C_DIS
LIN {X 0.131,Y -598.298,Z 982.308,A 0.000,B 0.000,C 90.000,E1 271.489} C_DIS
LIN {X -0.091,Y -591.329,Z 982.307,A 0.000,B 0.000,C 90.000,E1 271.203} C_DIS
LIN {X -0.026,Y -584.102,Z 982.305,A 0.000,B 0.000,C 90.000,E1 270.917} C_DIS
LIN {X -0.143,Y -578.148,Z 982.304,A 0.000,B 0.000,C 90.000,E1 270.745} C_DIS
LIN {X 0.229,Y -570.486,Z 982.303,A 0.000,B 0.000,C 90.000,E1 270.516} C_DIS
LIN {X 0.162,Y -564.735,Z 982.302,A 0.000,B 0.000,C 90.000,E1 270.401} C_DIS
LIN {X 0.063,Y -557.739,Z 982.302,A 0.000,B 0.000,C 90.000,E1 270.344} C_DIS
LIN {X 0.033,Y -545.986,Z 982.302,A 0.000,B 0.000,C 90.000,E1 270.344} C_DIS
LIN {X -0.018,Y -542.849,Z 982.301,A 0.000,B 0.000,C 90.000,E1 270.172} C_DIS
LIN {X -0.072,Y -542.780,Z 982.301,A 0.000,B 0.000,C 90.000,E1 270.172} C_DIS
LIN {X 0.202,Y -541.019,Z 982.288,A 0.000,B 0.000,C 90.000,E1 267.764} C_DIS
LIN {X -0.199,Y -539.791,Z 982.278,A 0.000,B 0.000,C 90.000,E1 266.102} C_DIS
LIN {X -0.070,Y -538.779,Z 982.270,A 0.000,B 0.000,C 90.000,E1 264.666} C_DIS
LIN {X 0.039,Y -537.857,Z 982.264,A 0.000,B 0.000,C 90.000,E1 263.514} C_DIS
LIN {X 0.237,Y -536.220,Z 982.255,A 0.000,B 0.000,C 90.000,E1 261.781} C_DIS
LIN {X -0.100,Y -534.784,Z 982.247,A 0.000,B 0.000,C 90.000,E1 260.387} C_DIS
LIN {X 0.163,Y -533.263,Z 982.239,A 0.000,B 0.000,C 90.000,E1 258.926} C_DIS
LIN {X -0.077,Y -531.387,Z 982.229,A 0.000,B 0.000,C 90.000,E1 257.229} C_DIS
LIN {X -0.186,Y -528.600,Z 982.216,A 0.000,B 0.000,C 90.000,E1 254.936} C_DIS
LIN {X -0.126,Y -526.494,Z 982.205,A 0.000,B 0.000,C 90.000,E1 252.906} C_DIS
LIN {X -0.122,Y -524.808,Z 982.197,A 0.000,B 0.000,C 90.000,E1 251.456} C_DIS
LIN {X -0.135,Y -523.324,Z 982.190,A 0.000,B 0.000,C 90.000,E1 250.296} C_DIS
LIN {X -0.007,Y -521.460,Z 982.182,A 0.000,B 0.000,C 90.000,E1 248.827} C_DIS
LIN {X 0.077,Y -519.610,Z 982.174,A 0.000,B 0.000,C 90.000,E1 247.358} C_DIS
LIN {X 0.036,Y -518.407,Z 982.169,A 0.000,B 0.000,C 90.000,E1 246.485} C_DIS
LIN {X -0.007,Y -516.235,Z 982.161,A 0.000,B 0.000,C 90.000,E1 245.025} C_DIS
LIN {X -0.083,Y -513.876,Z 982.153,A 0.000,B 0.000,C 90.000,E1 243.563} C_DIS
LIN {X 0.139,Y -512.044,Z 982.147,A 0.000,B 0.000,C 90.000,E1 242.359} C_DIS
LIN {X -0.243,Y -509.640,Z 982.138,A 0.000,B 0.000,C 90.000,E1 240.923} C_DIS
LIN {X -0.047,Y -507.547,Z 982.132,A 0.000,B 0.000,C 90.000,E1 239.715} C_DIS
LIN {X -0.139,Y -505.400,Z 982.125,A 0.000,B 0.000,C 90.000,E1 238.535} C_DIS
LIN {X -0.010,Y -502.945,Z 982.119,A 0.000,B 0.000,C 90.000,E1 237.327} C_DIS
LIN {X 0.229,Y -499.705,Z 982.110,A 0.000,B 0.000,C 90.000,E1 235.801} C_DIS
LIN {X -0.131,Y -495.573,Z 982.100,A 0.000,B 0.000,C 90.000,E1 234.036} C_DIS
LIN {X -0.289,Y -492.713,Z 982.093,A 0.000,B 0.000,C 90.000,E1 232.844} C_DIS
LIN {X 0.173,Y -488.418,Z 982.083,A 0.000,B 0.000,C 90.000,E1 230.964} C_DIS
LIN {X -0.050,Y -484.832,Z 982.075,A 0.000,B 0.000,C 90.000,E1 229.461} C_DIS
LIN {X -0.085,Y -479.864,Z 982.063,A 0.000,B 0.000,C 90.000,E1 227.310} C_DIS
LIN {X -0.040,Y -475.876,Z 982.052,A 0.000,B 0.000,C 90.000,E1 225.445} C_DIS
LIN {X 0.043,Y -473.219,Z 982.046,A 0.000,B 0.000,C 90.000,E1 224.190} C_DIS
LIN {X 0.179,Y -469.760,Z 982.037,A 0.000,B 0.000,C 90.000,E1 222.609} C_DIS
LIN {X -0.069,Y -466.286,Z 982.028,A 0.000,B 0.000,C 90.000,E1 221.067} C_DIS
LIN {X -0.285,Y -462.062,Z 982.018,A 0.000,B 0.000,C 90.000,E1 219.197} C_DIS
LIN {X 0.232,Y -456.375,Z 982.003,A 0.000,B 0.000,C 90.000,E1 216.583} C_DIS
LIN {X 0.149,Y -453.529,Z 981.996,A 0.000,B 0.000,C 90.000,E1 215.311} C_DIS
LIN {X 0.102,Y -450.011,Z 981.987,A 0.000,B 0.000,C 90.000,E1 213.706} C_DIS
LIN {X 0.116,Y -446.510,Z 981.978,A 0.000,B 0.000,C 90.000,E1 212.084} C_DIS
LIN {X 0.119,Y -442.335,Z 981.968,A 0.000,B 0.000,C 90.000,E1 210.129} C_DIS
LIN {X 0.097,Y -439.407,Z 981.960,A 0.000,B 0.000,C 90.000,E1 208.821} C_DIS
LIN {X 0.106,Y -433.647,Z 981.946,A 0.000,B 0.000,C 90.000,E1 206.181} C_DIS
LIN {X 0.142,Y -430.557,Z 981.938,A 0.000,B 0.000,C 90.000,E1 204.847} C_DIS
LIN {X -0.270,Y -425.931,Z 981.927,A 0.000,B 0.000,C 90.000,E1 202.898} C_DIS
LIN {X 0.158,Y -420.811,Z 981.914,A 0.000,B 0.000,C 90.000,E1 200.482} C_DIS
LIN {X -0.023,Y -416.514,Z 981.903,A 0.000,B 0.000,C 90.000,E1 198.471} C_DIS
LIN {X 0.106,Y -411.352,Z 981.887,A 0.000,B 0.000,C 90.000,E1 195.717} C_DIS
LIN {X 0.015,Y -408.251,Z 981.878,A 0.000,B 0.000,C 90.000,E1 194.008} C_DIS
LIN {X -0.132,Y -405.095,Z 981.868,A 0.000,B 0.000,C 90.000,E1 192.299} C_DIS
LIN {X -0.034,Y -401.793,Z 981.859,A 0.000,B 0.000,C 90.000,E1 190.546} C_DIS
LIN {X -0.061,Y -399.223,Z 981.851,A 0.000,B 0.000,C 90.000,E1 189.151} C_DIS
LIN {X 0.158,Y -395.559,Z 981.839,A 0.000,B 0.000,C 90.000,E1 187.011} C_DIS
LIN {X -0.025,Y -393.764,Z 981.831,A 0.000,B 0.000,C 90.000,E1 185.625} C_DIS
LIN {X 0.197,Y -393.125,Z 981.825,A 0.000,B 0.000,C 90.000,E1 184.531} C_DIS
LIN {X 0.066,Y -393.297,Z 981.821,A 0.000,B 0.000,C 90.000,E1 183.841} C_DIS
LIN {X -0.087,Y -394.300,Z 981.818,A 0.000,B 0.000,C 90.000,E1 183.154} C_DIS
LIN {X -0.166,Y -395.653,Z 981.815,A 0.000,B 0.000,C 90.000,E1 182.636} C_DIS
LIN {X 0.124,Y -397.251,Z 981.812,A 0.000,B 0.000,C 90.000,E1 182.178} C_DIS
LIN {X 0.063,Y -398.832,Z 981.810,A 0.000,B 0.000,C 90.000,E1 181.835} C_DIS
LIN {X 0.158,Y -401.487,Z 981.808,A 0.000,B 0.000,C 90.000,E1 181.375} C_DIS
LIN {X 0.178,Y -405.178,Z 981.805,A 0.000,B 0.000,C 90.000,E1 180.859} C_DIS
LIN {X -0.004,Y -412.256,Z 981.801,A 0.000,B 0.000,C 90.000,E1 180.115} C_DIS
LIN {X -0.110,Y -428.738,Z 981.792,A 0.000,B 0.000,C 90.000,E1 178.511} C_DIS
LIN {X -0.081,Y -434.668,Z 981.789,A 0.000,B 0.000,C 90.000,E1 177.936} C_DIS
LIN {X -0.159,Y -443.379,Z 981.784,A 0.000,B 0.000,C 90.000,E1 177.078} C_DIS
LIN {X -0.155,Y -453.364,Z 981.778,A 0.000,B 0.000,C 90.000,E1 176.045} C_DIS
LIN {X -0.180,Y -458.751,Z 981.775,A 0.000,B 0.000,C 90.000,E1 175.469} C_DIS
LIN {X 0.175,Y -464.120,Z 981.771,A 0.000,B 0.000,C 90.000,E1 174.837} C_DIS
LIN {X -0.131,Y -473.474,Z 981.766,A 0.000,B 0.000,C 90.000,E1 173.799} C_DIS
LIN {X 0.122,Y -479.865,Z 981.761,A 0.000,B 0.000,C 90.000,E1 172.996} C_DIS
LIN {X -0.084,Y -488.055,Z 981.755,A 0.000,B 0.000,C 90.000,E1 171.951} C_DIS
LIN {X -0.018,Y -494.996,Z 981.750,A 0.000,B 0.000,C 90.000,E1 171.027} C_DIS
LIN {X -0.043,Y -500.550,Z 981.746,A 0.000,B 0.000,C 90.000,E1 170.274} C_DIS
LIN {X 0.192,Y -508.774,Z 981.739,A 0.000,B 0.000,C 90.000,E1 169.050} C_DIS
LIN {X -0.137,Y -515.523,Z 981.734,A 0.000,B 0.000,C 90.000,E1 168.049} C_DIS
LIN {X -0.122,Y -519.369,Z 981.730,A 0.000,B 0.000,C 90.000,E1 167.465} C_DIS
LIN {X 0.195,Y -525.822,Z 981.725,A 0.000,B 0.000,C 90.000,E1 166.408} C_DIS
LIN {X -0.093,Y -532.900,Z 981.718,A 0.000,B 0.000,C 90.000,E1 165.283} C_DIS
LIN {X 0.235,Y -539.817,Z 981.712,A 0.000,B 0.000,C 90.000,E1 164.102} C_DIS
LIN {X -0.148,Y -548.010,Z 981.704,A 0.000,B 0.000,C 90.000,E1 162.725} C_DIS
LIN {X -0.070,Y -552.942,Z 981.699,A 0.000,B 0.000,C 90.000,E1 161.873} C_DIS
LIN {X -0.038,Y -562.963,Z 981.689,A 0.000,B 0.000,C 90.000,E1 160.061} C_DIS
LIN {X 0.150,Y -570.305,Z 981.682,A 0.000,B 0.000,C 90.000,E1 158.666} C_DIS
LIN {X -0.013,Y -575.803,Z 981.676,A 0.000,B 0.000,C 90.000,E1 157.592} C_DIS
LIN {X 0.217,Y -580.862,Z 981.670,A 0.000,B 0.000,C 90.000,E1 156.485} C_DIS
LIN {X 0.216,Y -585.683,Z 981.664,A 0.000,B 0.000,C 90.000,E1 155.409} C_DIS
LIN {X -0.276,Y -587.980,Z 981.661,A 0.000,B 0.000,C 90.000,E1 154.921} C_DIS
LIN {X 0.023,Y -590.115,Z 981.658,A 0.000,B 0.000,C 90.000,E1 154.357} C_DIS
LIN {X -0.034,Y -593.029,Z 981.653,A 0.000,B 0.000,C 90.000,E1 153.563} C_DIS
LIN {X 0.121,Y -596.662,Z 981.647,A 0.000,B 0.000,C 90.000,E1 152.487} C_DIS
LIN {X 0.071,Y -600.039,Z 981.641,A 0.000,B 0.000,C 90.000,E1 151.435} C_DIS
LIN {X 0.073,Y -603.175,Z 981.636,A 0.000,B 0.000,C 90.000,E1 150.383} C_DIS
LIN {X 0.054,Y -607.154,Z 981.628,A 0.000,B 0.000,C 90.000,E1 149.076} C_DIS
LIN {X -0.111,Y -611.057,Z 981.621,A 0.000,B 0.000,C 90.000,E1 147.788} C_DIS
LIN {X -0.172,Y -617.280,Z 981.609,A 0.000,B 0.000,C 90.000,E1 145.722} C_DIS
LIN {X -0.040,Y -622.632,Z 981.600,A 0.000,B 0.000,C 90.000,E1 143.909} C_DIS
LIN {X 0.230,Y -627.165,Z 981.591,A 0.000,B 0.000,C 90.000,E1 142.351} C_DIS
LIN {X 0.254,Y -630.214,Z 981.585,A 0.000,B 0.000,C 90.000,E1 141.331} C_DIS
LIN {X -0.034,Y -635.412,Z 981.576,A 0.000,B 0.000,C 90.000,E1 139.585} C_DIS
LIN {X -0.194,Y -640.434,Z 981.566,A 0.000,B 0.000,C 90.000,E1 137.838} C_DIS
LIN {X 0.259,Y -644.947,Z 981.557,A 0.000,B 0.000,C 90.000,E1 136.296} C_DIS
LIN {X -0.244,Y -651.233,Z 981.546,A 0.000,B 0.000,C 90.000,E1 134.352} C_DIS
LIN {X -0.153,Y -658.775,Z 981.534,A 0.000,B 0.000,C 90.000,E1 132.123} C_DIS
LIN {X 0.226,Y -665.044,Z 981.524,A 0.000,B 0.000,C 90.000,E1 130.378} C_DIS
LIN {X -0.182,Y -669.392,Z 981.518,A 0.000,B 0.000,C 90.000,E1 129.197} C_DIS
LIN {X 0.005,Y -674.251,Z 981.510,A 0.000,B 0.000,C 90.000,E1 127.729} C_DIS
LIN {X 0.272,Y -677.949,Z 981.503,A 0.000,B 0.000,C 90.000,E1 126.503} C_DIS
LIN {X -0.191,Y -682.252,Z 981.495,A 0.000,B 0.000,C 90.000,E1 125.105} C_DIS
LIN {X -0.391,Y -684.321,Z 981.491,A 0.000,B 0.000,C 90.000,E1 124.405} C_DIS
LIN {X 0.003,Y -686.895,Z 981.486,A 0.000,B 0.000,C 90.000,E1 123.420} C_DIS
LIN {X 0.121,Y -691.293,Z 981.477,A 0.000,B 0.000,C 90.000,E1 121.750} C_DIS
LIN {X 0.226,Y -693.597,Z 981.471,A 0.000,B 0.000,C 90.000,E1 120.797} C_DIS
LIN {X -0.247,Y -695.175,Z 981.467,A 0.000,B 0.000,C 90.000,E1 120.129} C_DIS
LIN {X -0.102,Y -696.610,Z 981.463,A 0.000,B 0.000,C 90.000,E1 119.411} C_DIS
LIN {X 0.059,Y -697.742,Z 981.459,A 0.000,B 0.000,C 90.000,E1 118.693} C_DIS
LIN {X 0.232,Y -698.574,Z 981.456,A 0.000,B 0.000,C 90.000,E1 117.975} C_DIS
LIN {X -0.346,Y -699.874,Z 981.448,A 0.000,B 0.000,C 90.000,E1 116.616} C_DIS
LIN {X 0.077,Y -700.764,Z 981.441,A 0.000,B 0.000,C 90.000,E1 115.412} C_DIS
LIN {X -0.033,Y -701.051,Z 981.437,A 0.000,B 0.000,C 90.000,E1 114.719} C_DIS
LIN {X -0.125,Y -701.112,Z 981.435,A 0.000,B 0.000,C 90.000,E1 114.259} C_DIS
LIN {X 0.133,Y -700.704,Z 981.432,A 0.000,B 0.000,C 90.000,E1 113.770} C_DIS
LIN {X -0.238,Y -700.375,Z 981.431,A 0.000,B 0.000,C 90.000,E1 113.567} C_DIS
LIN {X 0.019,Y -698.727,Z 981.428,A 0.000,B 0.000,C 90.000,E1 113.078} C_DIS
LIN {X 0.282,Y -697.575,Z 981.427,A 0.000,B 0.000,C 90.000,E1 112.823} C_DIS
LIN {X 0.270,Y -695.373,Z 981.426,A 0.000,B 0.000,C 90.000,E1 112.589} C_DIS
LIN {X -0.223,Y -691.685,Z 981.424,A 0.000,B 0.000,C 90.000,E1 112.280} C_DIS
LIN {X -0.075,Y -689.681,Z 981.423,A 0.000,B 0.000,C 90.000,E1 112.153} C_DIS
LIN {X 0.000,Y -684.974,Z 981.422,A 0.000,B 0.000,C 90.000,E1 111.972} C_DIS
LIN {X 0.143,Y -682.554,Z 981.422,A 0.000,B 0.000,C 90.000,E1 111.897} C_DIS
LIN {X 0.029,Y -675.870,Z 981.421,A 0.000,B 0.000,C 90.000,E1 111.770} C_DIS
LIN {X -0.150,Y -673.367,Z 981.421,A 0.000,B 0.000,C 90.000,E1 111.770} C_DIS
LIN {X -0.208,Y -669.496,Z 981.421,A 0.000,B 0.000,C 90.000,E1 111.770} C_DIS
LIN {X -0.239,Y -624.121,Z 981.421,A 0.000,B 0.000,C 90.000,E1 111.770} C_DIS
LIN {X 0.200,Y -617.090,Z 981.420,A 0.000,B 0.000,C 90.000,E1 111.589} C_DIS
LIN {X -0.056,Y -610.135,Z 981.419,A 0.000,B 0.000,C 90.000,E1 111.408} C_DIS
LIN {X 0.288,Y -603.338,Z 981.417,A 0.000,B 0.000,C 90.000,E1 111.099} C_DIS
LIN {X -0.014,Y -596.972,Z 981.416,A 0.000,B 0.000,C 90.000,E1 110.791} C_DIS
LIN {X 0.123,Y -590.016,Z 981.413,A 0.000,B 0.000,C 90.000,E1 110.301} C_DIS
LIN {X 0.029,Y -578.920,Z 981.408,A 0.000,B 0.000,C 90.000,E1 109.450} C_DIS
LIN {X 0.291,Y -574.530,Z 981.406,A 0.000,B 0.000,C 90.000,E1 109.087} C_DIS
LIN {X 0.051,Y -566.297,Z 981.403,A 0.000,B 0.000,C 90.000,E1 108.598} C_DIS
LIN {X 0.236,Y -551.494,Z 981.399,A 0.000,B 0.000,C 90.000,E1 107.819} C_DIS
LIN {X -0.178,Y -549.632,Z 981.398,A 0.000,B 0.000,C 90.000,E1 107.692} C_DIS
LIN {X -0.215,Y -549.607,Z 981.398,A 0.000,B 0.000,C 90.000,E1 107.692} C_DIS
LIN {X 0.042,Y -549.175,Z 981.397,A 0.000,B 0.000,C 90.000,E1 107.402} C_DIS
LIN {X 0.076,Y -549.498,Z 981.390,A 0.000,B 0.000,C 90.000,E1 106.134} C_DIS
LIN {X 0.097,Y -550.004,Z 981.383,A 0.000,B 0.000,C 90.000,E1 105.009} C_DIS
LIN {X -0.077,Y -551.039,Z 981.373,A 0.000,B 0.000,C 90.000,E1 103.063} C_DIS
LIN {X 0.142,Y -553.701,Z 981.355,A 0.000,B 0.000,C 90.000,E1 99.962} C_DIS
LIN {X 0.250,Y -555.460,Z 981.346,A 0.000,B 0.000,C 90.000,E1 98.276} C_DIS
LIN {X 0.242,Y -557.110,Z 981.337,A 0.000,B 0.000,C 90.000,E1 96.606} C_DIS
LIN {X 0.203,Y -558.202,Z 981.329,A 0.000,B 0.000,C 90.000,E1 95.220} C_DIS
LIN {X 0.125,Y -559.143,Z 981.321,A 0.000,B 0.000,C 90.000,E1 93.841} C_DIS
LIN {X 0.027,Y -559.947,Z 981.314,A 0.000,B 0.000,C 90.000,E1 92.465} C_DIS
LIN {X 0.135,Y -560.951,Z 981.303,A 0.000,B 0.000,C 90.000,E1 90.516} C_DIS
LIN {X 0.058,Y -561.501,Z 981.295,A 0.000,B 0.000,C 90.000,E1 89.141} C_DIS
LIN {X 0.002,Y -561.846,Z 981.288,A 0.000,B 0.000,C 90.000,E1 87.764} C_DIS
LIN {X 0.049,Y -562.187,Z 981.278,A 0.000,B 0.000,C 90.000,E1 86.102} C_DIS
LIN {X 0.267,Y -562.428,Z 981.268,A 0.000,B 0.000,C 90.000,E1 84.147} C_DIS
LIN {X 0.145,Y -562.809,Z 981.255,A 0.000,B 0.000,C 90.000,E1 81.951} C_DIS
LIN {X -0.040,Y -563.359,Z 981.245,A 0.000,B 0.000,C 90.000,E1 80.038} C_DIS
LIN {X 0.040,Y -564.354,Z 981.232,A 0.000,B 0.000,C 90.000,E1 77.825} C_DIS
LIN {X 0.306,Y -566.047,Z 981.217,A 0.000,B 0.000,C 90.000,E1 75.046} C_DIS
LIN {X -0.251,Y -567.553,Z 981.205,A 0.000,B 0.000,C 90.000,E1 72.906} C_DIS
LIN {X -0.011,Y -568.480,Z 981.197,A 0.000,B 0.000,C 90.000,E1 71.511} C_DIS
LIN {X 0.059,Y -569.356,Z 981.190,A 0.000,B 0.000,C 90.000,E1 70.134} C_DIS
LIN {X -0.006,Y -570.077,Z 981.182,A 0.000,B 0.000,C 90.000,E1 68.773} C_DIS
LIN {X 0.126,Y -570.625,Z 981.176,A 0.000,B 0.000,C 90.000,E1 67.667} C_DIS
LIN {X -0.085,Y -571.247,Z 981.167,A 0.000,B 0.000,C 90.000,E1 66.049} C_DIS
LIN {X 0.114,Y -571.710,Z 981.159,A 0.000,B 0.000,C 90.000,E1 64.665} C_DIS
LIN {X -0.106,Y -572.139,Z 981.150,A 0.000,B 0.000,C 90.000,E1 63.050} C_DIS
LIN {X -0.147,Y -572.451,Z 981.143,A 0.000,B 0.000,C 90.000,E1 61.691} C_DIS
LIN {X -0.071,Y -572.659,Z 981.134,A 0.000,B 0.000,C 90.000,E1 60.049} C_DIS
LIN {X 0.169,Y -572.811,Z 981.126,A 0.000,B 0.000,C 90.000,E1 58.663} C_DIS
LIN {X 0.086,Y -572.986,Z 981.120,A 0.000,B 0.000,C 90.000,E1 57.582} C_DIS
LIN {X 0.141,Y -573.055,Z 981.112,A 0.000,B 0.000,C 90.000,E1 56.215} C_DIS
LIN {X 0.048,Y -573.054,Z 981.106,A 0.000,B 0.000,C 90.000,E1 55.135} C_DIS
LIN {X 0.002,Y -572.915,Z 981.102,A 0.000,B 0.000,C 90.000,E1 54.322} C_DIS
LIN {X 0.052,Y -572.374,Z 981.093,A 0.000,B 0.000,C 90.000,E1 52.683} C_DIS
LIN {X -0.196,Y -571.780,Z 981.087,A 0.000,B 0.000,C 90.000,E1 51.618} C_DIS
LIN {X -0.103,Y -570.942,Z 981.081,A 0.000,B 0.000,C 90.000,E1 50.517} C_DIS
LIN {X -0.154,Y -570.267,Z 981.076,A 0.000,B 0.000,C 90.000,E1 49.703} C_DIS
LIN {X -0.148,Y -569.100,Z 981.070,A 0.000,B 0.000,C 90.000,E1 48.609} C_DIS
LIN {X 0.086,Y -568.457,Z 981.067,A 0.000,B 0.000,C 90.000,E1 48.038} C_DIS
LIN {X 0.067,Y -566.758,Z 981.061,A 0.000,B 0.000,C 90.000,E1 46.944} C_DIS
LIN {X -0.068,Y -565.334,Z 981.056,A 0.000,B 0.000,C 90.000,E1 46.134} C_DIS
LIN {X -0.214,Y -563.714,Z 981.052,A 0.000,B 0.000,C 90.000,E1 45.324} C_DIS
LIN {X 0.097,Y -561.307,Z 981.046,A 0.000,B 0.000,C 90.000,E1 44.190} C_DIS
LIN {X -0.018,Y -558.289,Z 981.039,A 0.000,B 0.000,C 90.000,E1 43.095} C_DIS
LIN {X 0.098,Y -556.644,Z 981.036,A 0.000,B 0.000,C 90.000,E1 42.528} C_DIS
LIN {X 0.263,Y -553.855,Z 981.032,A 0.000,B 0.000,C 90.000,E1 41.676} C_DIS
LIN {X -0.026,Y -551.824,Z 981.029,A 0.000,B 0.000,C 90.000,E1 41.148} C_DIS
LIN {X 0.084,Y -548.472,Z 981.024,A 0.000,B 0.000,C 90.000,E1 40.297} C_DIS
LIN {X -0.200,Y -544.766,Z 981.019,A 0.000,B 0.000,C 90.000,E1 39.483} C_DIS
LIN {X 0.054,Y -541.390,Z 981.015,A 0.000,B 0.000,C 90.000,E1 38.749} C_DIS
LIN {X 0.116,Y -537.021,Z 981.011,A 0.000,B 0.000,C 90.000,E1 37.890} C_DIS
LIN {X 0.135,Y -532.414,Z 981.006,A 0.000,B 0.000,C 90.000,E1 37.030} C_DIS
LIN {X 0.104,Y -527.557,Z 981.001,A 0.000,B 0.000,C 90.000,E1 36.171} C_DIS
LIN {X 0.223,Y -525.029,Z 980.999,A 0.000,B 0.000,C 90.000,E1 35.724} C_DIS
LIN {X -0.073,Y -518.810,Z 980.993,A 0.000,B 0.000,C 90.000,E1 34.739} C_DIS
LIN {X -0.124,Y -512.908,Z 980.988,A 0.000,B 0.000,C 90.000,E1 33.865} C_DIS
LIN {X -0.101,Y -509.821,Z 980.986,A 0.000,B 0.000,C 90.000,E1 33.420} C_DIS
LIN {X -0.055,Y -504.343,Z 980.982,A 0.000,B 0.000,C 90.000,E1 32.673} C_DIS
LIN {X 0.065,Y -500.796,Z 980.979,A 0.000,B 0.000,C 90.000,E1 32.212} C_DIS
LIN {X 0.165,Y -497.130,Z 980.977,A 0.000,B 0.000,C 90.000,E1 31.750} C_DIS
LIN {X -0.066,Y -491.861,Z 980.973,A 0.000,B 0.000,C 90.000,E1 31.180} C_DIS
LIN {X 0.112,Y -487.769,Z 980.971,A 0.000,B 0.000,C 90.000,E1 30.718} C_DIS
LIN {X 0.260,Y -482.167,Z 980.968,A 0.000,B 0.000,C 90.000,E1 30.129} C_DIS
LIN {X -0.167,Y -472.127,Z 980.962,A 0.000,B 0.000,C 90.000,E1 29.205} C_DIS
LIN {X 0.153,Y -466.265,Z 980.959,A 0.000,B 0.000,C 90.000,E1 28.615} C_DIS
LIN {X -0.196,Y -455.828,Z 980.954,A 0.000,B 0.000,C 90.000,E1 27.719} C_DIS
LIN {X 0.050,Y -445.469,Z 980.949,A 0.000,B 0.000,C 90.000,E1 26.796} C_DIS
LIN {X -0.015,Y -423.133,Z 980.938,A 0.000,B 0.000,C 90.000,E1 24.847} C_DIS
LIN {X -0.041,Y -410.165,Z 980.931,A 0.000,B 0.000,C 90.000,E1 23.590} C_DIS
LIN {X -0.004,Y -401.548,Z 980.926,A 0.000,B 0.000,C 90.000,E1 22.695} C_DIS
LIN {X 0.183,Y -397.616,Z 980.924,A 0.000,B 0.000,C 90.000,E1 22.206} C_DIS
LIN {X 0.209,Y -395.226,Z 980.922,A 0.000,B 0.000,C 90.000,E1 21.897} C_DIS
LIN {X -0.049,Y -392.080,Z 980.919,A 0.000,B 0.000,C 90.000,E1 21.408} C_DIS
LIN {X 0.003,Y -390.980,Z 980.917,A 0.000,B 0.000,C 90.000,E1 21.046} C_DIS
LIN {X 0.145,Y -389.971,Z 980.913,A 0.000,B 0.000,C 90.000,E1 20.301} C_DIS
LIN {X -0.114,Y -389.961,Z 980.910,A 0.000,B 0.000,C 90.000,E1 19.758} C_DIS
LIN {X -0.044,Y -394.769,Z 980.882,A 0.000,B 0.000,C 90.000,E1 14.773} C_DIS
LIN {X 0.009,Y -398.953,Z 980.864,A 0.000,B 0.000,C 90.000,E1 11.591} C_DIS
LIN {X -0.091,Y -404.075,Z 980.847,A 0.000,B 0.000,C 90.000,E1 8.454} C_DIS
LIN {X -0.129,Y -409.304,Z 980.832,A 0.000,B 0.000,C 90.000,E1 5.682} C_DIS
LIN {X -0.082,Y -415.126,Z 980.816,A 0.000,B 0.000,C 90.000,E1 2.922} C_DIS
LIN {X -0.015,Y -418.180,Z 980.809,A 0.000,B 0.000,C 90.000,E1 1.547} C_DIS
LIN {X 0.048,Y -420.463,Z 980.804,A 0.000,B 0.000,C 90.000,E1 0.688} C_DIS
LIN {X 0.000,Y -423.162,Z 980.800,A 0.000,B 0.000,C 90.000,E1 360.000} C_DIS
LIN {X 0.184,Y -425.476,Z 980.798,A 0.000,B 0.000,C 90.000,E1 359.599} C_DIS
LIN {X 0.208,Y -426.653,Z 980.797,A 0.000,B 0.000,C 90.000,E1 359.427} C_DIS
LIN {X -0.175,Y -428.626,Z 980.796,A 0.000,B 0.000,C 90.000,E1 359.255} C_DIS
LIN {X -0.071,Y -430.357,Z 980.795,A 0.000,B 0.000,C 90.000,E1 359.083} C_DIS
LIN {X -0.026,Y -434.024,Z 980.793,A 0.000,B 0.000,C 90.000,E1 358.797} C_DIS
LIN {X -0.088,Y -453.837,Z 980.787,A 0.000,B 0.000,C 90.000,E1 357.707} C_DIS
LIN {X -0.141,Y -470.636,Z 980.782,A 0.000,B 0.000,C 90.000,E1 356.788} C_DIS
LIN {X 0.199,Y -482.265,Z 980.779,A 0.000,B 0.000,C 90.000,E1 356.102} C_DIS
LIN {X -0.016,Y -493.663,Z 980.775,A 0.000,B 0.000,C 90.000,E1 355.469} C_DIS
LIN {X 0.085,Y -504.983,Z 980.771,A 0.000,B 0.000,C 90.000,E1 354.780} C_DIS
LIN {X 0.208,Y -512.961,Z 980.768,A 0.000,B 0.000,C 90.000,E1 354.261} C_DIS
LIN {X 0.210,Y -520.660,Z 980.765,A 0.000,B 0.000,C 90.000,E1 353.742} C_DIS
LIN {X -0.021,Y -528.266,Z 980.762,A 0.000,B 0.000,C 90.000,E1 353.223} C_DIS
LIN {X 0.100,Y -532.575,Z 980.760,A 0.000,B 0.000,C 90.000,E1 352.875} C_DIS
LIN {X -0.032,Y -538.342,Z 980.758,A 0.000,B 0.000,C 90.000,E1 352.413} C_DIS
LIN {X 0.169,Y -543.972,Z 980.755,A 0.000,B 0.000,C 90.000,E1 351.894} C_DIS
LIN {X 0.148,Y -550.513,Z 980.752,A 0.000,B 0.000,C 90.000,E1 351.254} C_DIS
LIN {X -0.047,Y -555.591,Z 980.749,A 0.000,B 0.000,C 90.000,E1 350.735} C_DIS
LIN {X 0.011,Y -561.403,Z 980.745,A 0.000,B 0.000,C 90.000,E1 350.038} C_DIS
LIN {X 0.198,Y -566.569,Z 980.741,A 0.000,B 0.000,C 90.000,E1 349.342} C_DIS
LIN {X -0.012,Y -570.495,Z 980.738,A 0.000,B 0.000,C 90.000,E1 348.814} C_DIS
LIN {X 0.126,Y -574.913,Z 980.734,A 0.000,B 0.000,C 90.000,E1 348.117} C_DIS
LIN {X -0.028,Y -578.188,Z 980.731,A 0.000,B 0.000,C 90.000,E1 347.589} C_DIS
LIN {X -0.136,Y -584.268,Z 980.725,A 0.000,B 0.000,C 90.000,E1 346.520} C_DIS
LIN {X 0.113,Y -587.818,Z 980.721,A 0.000,B 0.000,C 90.000,E1 345.825} C_DIS
LIN {X -0.162,Y -594.475,Z 980.714,A 0.000,B 0.000,C 90.000,E1 344.519} C_DIS
LIN {X -0.158,Y -600.653,Z 980.707,A 0.000,B 0.000,C 90.000,E1 343.196} C_DIS
LIN {X -0.203,Y -603.616,Z 980.703,A 0.000,B 0.000,C 90.000,E1 342.543} C_DIS
LIN {X -0.052,Y -609.084,Z 980.696,A 0.000,B 0.000,C 90.000,E1 341.221} C_DIS
LIN {X 0.129,Y -612.197,Z 980.691,A 0.000,B 0.000,C 90.000,E1 340.423} C_DIS
LIN {X 0.094,Y -616.067,Z 980.686,A 0.000,B 0.000,C 90.000,E1 339.390} C_DIS
LIN {X 0.082,Y -620.480,Z 980.678,A 0.000,B 0.000,C 90.000,E1 338.103} C_DIS
LIN {X -0.196,Y -624.567,Z 980.671,A 0.000,B 0.000,C 90.000,E1 336.847} C_DIS
LIN {X 0.174,Y -628.335,Z 980.664,A 0.000,B 0.000,C 90.000,E1 335.537} C_DIS
LIN {X -0.001,Y -631.154,Z 980.659,A 0.000,B 0.000,C 90.000,E1 334.537} C_DIS
LIN {X 0.169,Y -634.253,Z 980.652,A 0.000,B 0.000,C 90.000,E1 333.256} C_DIS
LIN {X 0.296,Y -636.008,Z 980.647,A 0.000,B 0.000,C 90.000,E1 332.487} C_DIS
LIN {X 0.031,Y -639.174,Z 980.639,A 0.000,B 0.000,C 90.000,E1 331.001} C_DIS
LIN {X 0.071,Y -641.604,Z 980.632,A 0.000,B 0.000,C 90.000,E1 329.744} C_DIS
LIN {X 0.027,Y -643.006,Z 980.628,A 0.000,B 0.000,C 90.000,E1 328.997} C_DIS
LIN {X 0.128,Y -644.974,Z 980.621,A 0.000,B 0.000,C 90.000,E1 327.740} C_DIS
LIN {X -0.008,Y -646.331,Z 980.615,A 0.000,B 0.000,C 90.000,E1 326.755} C_DIS
LIN {X 0.060,Y -647.582,Z 980.610,A 0.000,B 0.000,C 90.000,E1 325.754} C_DIS
LIN {X -0.034,Y -648.538,Z 980.604,A 0.000,B 0.000,C 90.000,E1 324.769} C_DIS
LIN {X -0.166,Y -649.131,Z 980.600,A 0.000,B 0.000,C 90.000,E1 324.036} C_DIS
LIN {X -0.233,Y -649.861,Z 980.595,A 0.000,B 0.000,C 90.000,E1 323.050} C_DIS
LIN {X 0.138,Y -650.554,Z 980.588,A 0.000,B 0.000,C 90.000,E1 321.778} C_DIS
LIN {X -0.096,Y -651.147,Z 980.581,A 0.000,B 0.000,C 90.000,E1 320.561} C_DIS
LIN {X -0.346,Y -651.886,Z 980.571,A 0.000,B 0.000,C 90.000,E1 318.852} C_DIS
LIN {X -0.303,Y -653.519,Z 980.558,A 0.000,B 0.000,C 90.000,E1 316.377} C_DIS
LIN {X -0.086,Y -654.631,Z 980.549,A 0.000,B 0.000,C 90.000,E1 314.879} C_DIS
LIN {X 0.080,Y -656.203,Z 980.538,A 0.000,B 0.000,C 90.000,E1 312.894} C_DIS
LIN {X -0.058,Y -657.160,Z 980.532,A 0.000,B 0.000,C 90.000,E1 311.676} C_DIS
LIN {X -0.174,Y -658.039,Z 980.525,A 0.000,B 0.000,C 90.000,E1 310.458} C_DIS
LIN {X -0.230,Y -658.949,Z 980.517,A 0.000,B 0.000,C 90.000,E1 308.991} C_DIS
LIN {X 0.214,Y -659.714,Z 980.507,A 0.000,B 0.000,C 90.000,E1 307.237} C_DIS
LIN {X -0.280,Y -659.977,Z 980.504,A 0.000,B 0.000,C 90.000,E1 306.790} C_DIS
LIN {X 0.304,Y -660.257,Z 980.495,A 0.000,B 0.000,C 90.000,E1 305.025} C_DIS
LIN {X 0.045,Y -660.600,Z 980.487,A 0.000,B 0.000,C 90.000,E1 303.579} C_DIS
LIN {X 0.067,Y -661.697,Z 980.473,A 0.000,B 0.000,C 90.000,E1 301.131} C_DIS
LIN {X 0.039,Y -668.213,Z 980.443,A 0.000,B 0.000,C 90.000,E1 295.771} C_DIS
LIN {X -0.057,Y -670.322,Z 980.437,A 0.000,B 0.000,C 90.000,E1 294.567} C_DIS
LIN {X 0.054,Y -671.886,Z 980.431,A 0.000,B 0.000,C 90.000,E1 293.590} C_DIS
LIN {X -0.325,Y -672.851,Z 980.427,A 0.000,B 0.000,C 90.000,E1 292.898} C_DIS
LIN {X 0.011,Y -673.320,Z 980.424,A 0.000,B 0.000,C 90.000,E1 292.386} C_DIS
LIN {X 0.092,Y -673.242,Z 980.422,A 0.000,B 0.000,C 90.000,E1 291.897} C_DIS
LIN {X 0.009,Y -673.121,Z 980.420,A 0.000,B 0.000,C 90.000,E1 291.663} C_DIS
LIN {X 0.095,Y -672.096,Z 980.418,A 0.000,B 0.000,C 90.000,E1 291.173} C_DIS
LIN {X 0.256,Y -671.330,Z 980.416,A 0.000,B 0.000,C 90.000,E1 290.918} C_DIS
LIN {X 0.176,Y -669.639,Z 980.415,A 0.000,B 0.000,C 90.000,E1 290.684} C_DIS
LIN {X 0.327,Y -667.360,Z 980.414,A 0.000,B 0.000,C 90.000,E1 290.429} C_DIS
LIN {X -0.362,Y -664.817,Z 980.412,A 0.000,B 0.000,C 90.000,E1 290.248} C_DIS
LIN {X -0.206,Y -658.551,Z 980.410,A 0.000,B 0.000,C 90.000,E1 289.812} C_DIS
LIN {X -0.195,Y -652.498,Z 980.408,A 0.000,B 0.000,C 90.000,E1 289.450} C_DIS
LIN {X -0.287,Y -649.510,Z 980.407,A 0.000,B 0.000,C 90.000,E1 289.214} C_DIS
LIN {X -0.326,Y -649.480,Z 980.407,A 0.000,B 0.000,C 90.000,E1 289.214} C_DIS
LIN {X -0.121,Y -649.293,Z 980.406,A 0.000,B 0.000,C 90.000,E1 289.141} C_DIS
LIN {X -0.159,Y -649.282,Z 980.406,A 0.000,B 0.000,C 90.000,E1 289.141} C_DIS
LIN {X 0.151,Y -650.418,Z 980.404,A 0.000,B 0.000,C 90.000,E1 288.725} C_DIS
LIN {X 0.047,Y -652.309,Z 980.402,A 0.000,B 0.000,C 90.000,E1 288.362} C_DIS
LIN {X 0.009,Y -657.621,Z 980.397,A 0.000,B 0.000,C 90.000,E1 287.511} C_DIS
LIN {X -0.319,Y -661.752,Z 980.393,A 0.000,B 0.000,C 90.000,E1 286.804} C_DIS
LIN {X 0.174,Y -664.868,Z 980.390,A 0.000,B 0.000,C 90.000,E1 286.150} C_DIS
LIN {X 0.103,Y -667.608,Z 980.386,A 0.000,B 0.000,C 90.000,E1 285.426} C_DIS
LIN {X -0.052,Y -669.060,Z 980.383,A 0.000,B 0.000,C 90.000,E1 284.954} C_DIS
LIN {X -0.266,Y -670.671,Z 980.379,A 0.000,B 0.000,C 90.000,E1 284.245} C_DIS
LIN {X 0.128,Y -672.069,Z 980.374,A 0.000,B 0.000,C 90.000,E1 283.244} C_DIS
LIN {X -0.056,Y -672.699,Z 980.370,A 0.000,B 0.000,C 90.000,E1 282.535} C_DIS
LIN {X -0.179,Y -672.876,Z 980.367,A 0.000,B 0.000,C 90.000,E1 282.063} C_DIS
LIN {X 0.293,Y -672.748,Z 980.363,A 0.000,B 0.000,C 90.000,E1 281.299} C_DIS
LIN {X 0.036,Y -672.507,Z 980.360,A 0.000,B 0.000,C 90.000,E1 280.838} C_DIS
LIN {X -0.093,Y -671.981,Z 980.358,A 0.000,B 0.000,C 90.000,E1 280.366} C_DIS
LIN {X -0.348,Y -671.256,Z 980.355,A 0.000,B 0.000,C 90.000,E1 279.905} C_DIS
LIN {X 0.169,Y -670.271,Z 980.352,A 0.000,B 0.000,C 90.000,E1 279.378} C_DIS
LIN {X -0.015,Y -669.686,Z 980.351,A 0.000,B 0.000,C 90.000,E1 279.151} C_DIS
LIN {X -0.173,Y -668.227,Z 980.348,A 0.000,B 0.000,C 90.000,E1 278.681} C_DIS
LIN {X 0.032,Y -665.478,Z 980.344,A 0.000,B 0.000,C 90.000,E1 277.936} C_DIS
LIN {X -0.063,Y -664.476,Z 980.343,A 0.000,B 0.000,C 90.000,E1 277.701} C_DIS
LIN {X -0.257,Y -662.659,Z 980.341,A 0.000,B 0.000,C 90.000,E1 277.352} C_DIS
LIN {X 0.193,Y -660.657,Z 980.339,A 0.000,B 0.000,C 90.000,E1 276.947} C_DIS
LIN {X -0.125,Y -657.608,Z 980.336,A 0.000,B 0.000,C 90.000,E1 276.486} C_DIS
LIN {X 0.084,Y -653.101,Z 980.333,A 0.000,B 0.000,C 90.000,E1 275.853} C_DIS
LIN {X -0.279,Y -649.095,Z 980.330,A 0.000,B 0.000,C 90.000,E1 275.391} C_DIS
LIN {X -0.139,Y -643.515,Z 980.326,A 0.000,B 0.000,C 90.000,E1 274.759} C_DIS
LIN {X 0.052,Y -638.668,Z 980.324,A 0.000,B 0.000,C 90.000,E1 274.245} C_DIS
LIN {X -0.192,Y -633.539,Z 980.321,A 0.000,B 0.000,C 90.000,E1 273.784} C_DIS
LIN {X -0.308,Y -626.685,Z 980.318,A 0.000,B 0.000,C 90.000,E1 273.212} C_DIS
LIN {X -0.213,Y -622.219,Z 980.316,A 0.000,B 0.000,C 90.000,E1 272.865} C_DIS
LIN {X 0.270,Y -616.439,Z 980.314,A 0.000,B 0.000,C 90.000,E1 272.407} C_DIS
LIN {X 0.117,Y -611.999,Z 980.312,A 0.000,B 0.000,C 90.000,E1 272.121} C_DIS
LIN {X 0.047,Y -603.835,Z 980.309,A 0.000,B 0.000,C 90.000,E1 271.661} C_DIS
LIN {X 0.123,Y -597.164,Z 980.307,A 0.000,B 0.000,C 90.000,E1 271.318} C_DIS
LIN {X -0.050,Y -590.043,Z 980.306,A 0.000,B 0.000,C 90.000,E1 271.031} C_DIS
LIN {X 0.222,Y -584.882,Z 980.305,A 0.000,B 0.000,C 90.000,E1 270.802} C_DIS
LIN {X 0.189,Y -577.280,Z 980.303,A 0.000,B 0.000,C 90.000,E1 270.573} C_DIS
LIN {X -0.117,Y -571.656,Z 980.303,A 0.000,B 0.000,C 90.000,E1 270.458} C_DIS
LIN {X -0.250,Y -565.718,Z 980.302,A 0.000,B 0.000,C 90.000,E1 270.344} C_DIS
LIN {X -0.063,Y -563.114,Z 980.302,A 0.000,B 0.000,C 90.000,E1 270.286} C_DIS
LIN {X 0.023,Y -557.791,Z 980.301,A 0.000,B 0.000,C 90.000,E1 270.229} C_DIS
LIN {X -0.010,Y -546.195,Z 980.301,A 0.000,B 0.000,C 90.000,E1 270.229} C_DIS
LIN {X -0.184,Y -542.839,Z 980.300,A 0.000,B 0.000,C 90.000,E1 270.057} C_DIS
LIN {X -0.238,Y -542.763,Z 980.300,A 0.000,B 0.000,C 90.000,E1 270.057} C_DIS
LIN {X -0.240,Y -542.330,Z 980.298,A 0.000,B 0.000,C 90.000,E1 269.599} C_DIS
LIN {X -0.066,Y -541.153,Z 980.288,A 0.000,B 0.000,C 90.000,E1 267.879} C_DIS
LIN {X 0.127,Y -539.751,Z 980.277,A 0.000,B 0.000,C 90.000,E1 265.869} C_DIS
LIN {X 0.264,Y -538.724,Z 980.269,A 0.000,B 0.000,C 90.000,E1 264.432} C_DIS
LIN {X -0.214,Y -538.044,Z 980.265,A 0.000,B 0.000,C 90.000,E1 263.628} C_DIS
LIN {X -0.007,Y -536.450,Z 980.255,A 0.000,B 0.000,C 90.000,E1 261.894} C_DIS
LIN {X 0.192,Y -534.998,Z 980.247,A 0.000,B 0.000,C 90.000,E1 260.443} C_DIS
LIN {X -0.216,Y -533.807,Z 980.241,A 0.000,B 0.000,C 90.000,E1 259.342} C_DIS
LIN {X 0.110,Y -531.578,Z 980.230,A 0.000,B 0.000,C 90.000,E1 257.297} C_DIS
LIN {X 0.128,Y -528.775,Z 980.217,A 0.000,B 0.000,C 90.000,E1 254.991} C_DIS
LIN {X 0.016,Y -527.268,Z 980.209,A 0.000,B 0.000,C 90.000,E1 253.559} C_DIS
LIN {X -0.125,Y -525.716,Z 980.201,A 0.000,B 0.000,C 90.000,E1 252.127} C_DIS
LIN {X -0.138,Y -523.940,Z 980.193,A 0.000,B 0.000,C 90.000,E1 250.678} C_DIS
LIN {X 0.146,Y -521.651,Z 980.183,A 0.000,B 0.000,C 90.000,E1 248.901} C_DIS
LIN {X -0.253,Y -519.805,Z 980.175,A 0.000,B 0.000,C 90.000,E1 247.486} C_DIS
LIN {X -0.293,Y -518.623,Z 980.170,A 0.000,B 0.000,C 90.000,E1 246.613} C_DIS
LIN {X -0.201,Y -515.971,Z 980.160,A 0.000,B 0.000,C 90.000,E1 244.845} C_DIS
LIN {X 0.174,Y -513.645,Z 980.152,A 0.000,B 0.000,C 90.000,E1 243.332} C_DIS
LIN {X -0.176,Y -512.260,Z 980.147,A 0.000,B 0.000,C 90.000,E1 242.487} C_DIS
LIN {X -0.107,Y -509.873,Z 980.139,A 0.000,B 0.000,C 90.000,E1 241.001} C_DIS
LIN {X -0.279,Y -507.281,Z 980.131,A 0.000,B 0.000,C 90.000,E1 239.537} C_DIS
LIN {X -0.117,Y -505.037,Z 980.124,A 0.000,B 0.000,C 90.000,E1 238.329} C_DIS
LIN {X 0.008,Y -502.535,Z 980.117,A 0.000,B 0.000,C 90.000,E1 237.120} C_DIS
LIN {X -0.051,Y -499.972,Z 980.111,A 0.000,B 0.000,C 90.000,E1 235.928} C_DIS
LIN {X -0.132,Y -495.170,Z 980.099,A 0.000,B 0.000,C 90.000,E1 233.829} C_DIS
LIN {X 0.001,Y -492.246,Z 980.092,A 0.000,B 0.000,C 90.000,E1 232.603} C_DIS
LIN {X -0.069,Y -488.756,Z 980.084,A 0.000,B 0.000,C 90.000,E1 231.090} C_DIS
LIN {X 0.093,Y -485.171,Z 980.075,A 0.000,B 0.000,C 90.000,E1 229.542} C_DIS
LIN {X 0.063,Y -480.183,Z 980.063,A 0.000,B 0.000,C 90.000,E1 227.391} C_DIS
LIN {X -0.226,Y -476.171,Z 980.053,A 0.000,B 0.000,C 90.000,E1 225.567} C_DIS
LIN {X 0.299,Y -472.805,Z 980.044,A 0.000,B 0.000,C 90.000,E1 223.947} C_DIS
LIN {X 0.188,Y -468.657,Z 980.034,A 0.000,B 0.000,C 90.000,E1 222.081} C_DIS
LIN {X -0.144,Y -465.900,Z 980.027,A 0.000,B 0.000,C 90.000,E1 220.862} C_DIS
LIN {X -0.111,Y -462.377,Z 980.018,A 0.000,B 0.000,C 90.000,E1 219.277} C_DIS
LIN {X 0.050,Y -456.646,Z 980.004,A 0.000,B 0.000,C 90.000,E1 216.710} C_DIS
LIN {X 0.061,Y -453.098,Z 979.995,A 0.000,B 0.000,C 90.000,E1 215.105} C_DIS
LIN {X 0.008,Y -449.583,Z 979.986,A 0.000,B 0.000,C 90.000,E1 213.499} C_DIS
LIN {X 0.014,Y -446.083,Z 979.977,A 0.000,B 0.000,C 90.000,E1 211.878} C_DIS
LIN {X -0.048,Y -442.611,Z 979.968,A 0.000,B 0.000,C 90.000,E1 210.256} C_DIS
LIN {X -0.066,Y -439.719,Z 979.961,A 0.000,B 0.000,C 90.000,E1 208.949} C_DIS
LIN {X 0.131,Y -434.633,Z 979.948,A 0.000,B 0.000,C 90.000,E1 206.616} C_DIS
LIN {X -0.027,Y -432.455,Z 979.943,A 0.000,B 0.000,C 90.000,E1 205.643} C_DIS
LIN {X 0.178,Y -428.545,Z 979.933,A 0.000,B 0.000,C 90.000,E1 203.951} C_DIS
LIN {X 0.073,Y -422.566,Z 979.918,A 0.000,B 0.000,C 90.000,E1 201.280} C_DIS
LIN {X -0.063,Y -418.240,Z 979.907,A 0.000,B 0.000,C 90.000,E1 199.268} C_DIS
LIN {X -0.122,Y -412.239,Z 979.890,A 0.000,B 0.000,C 90.000,E1 196.205} C_DIS
LIN {X -0.084,Y -409.112,Z 979.880,A 0.000,B 0.000,C 90.000,E1 194.481} C_DIS
LIN {X -0.114,Y -405.297,Z 979.869,A 0.000,B 0.000,C 90.000,E1 192.411} C_DIS
LIN {X -0.017,Y -401.982,Z 979.859,A 0.000,B 0.000,C 90.000,E1 190.658} C_DIS
LIN {X -0.044,Y -399.395,Z 979.852,A 0.000,B 0.000,C 90.000,E1 189.265} C_DIS
LIN {X 0.108,Y -394.563,Z 979.836,A 0.000,B 0.000,C 90.000,E1 186.429} C_DIS
LIN {X -0.011,Y -393.612,Z 979.832,A 0.000,B 0.000,C 90.000,E1 185.739} C_DIS
LIN {X -0.182,Y -392.769,Z 979.826,A 0.000,B 0.000,C 90.000,E1 184.702} C_DIS
LIN {X 0.075,Y -392.523,Z 979.822,A 0.000,B 0.000,C 90.000,E1 183.955} C_DIS
LIN {X -0.005,Y -392.668,Z 979.820,A 0.000,B 0.000,C 90.000,E1 183.612} C_DIS
LIN {X -0.142,Y -393.634,Z 979.816,A 0.000,B 0.000,C 90.000,E1 182.922} C_DIS
LIN {X 0.104,Y -395.551,Z 979.812,A 0.000,B 0.000,C 90.000,E1 182.178} C_DIS
LIN {X 0.035,Y -396.930,Z 979.810,A 0.000,B 0.000,C 90.000,E1 181.835} C_DIS
LIN {X -0.015,Y -398.643,Z 979.808,A 0.000,B 0.000,C 90.000,E1 181.489} C_DIS
LIN {X 0.094,Y -401.328,Z 979.806,A 0.000,B 0.000,C 90.000,E1 181.031} C_DIS
LIN {X 0.071,Y -404.864,Z 979.803,A 0.000,B 0.000,C 90.000,E1 180.573} C_DIS
LIN {X 0.036,Y -410.643,Z 979.800,A 0.000,B 0.000,C 90.000,E1 179.943} C_DIS
LIN {X -0.163,Y -429.884,Z 979.789,A 0.000,B 0.000,C 90.000,E1 178.108} C_DIS
LIN {X -0.103,Y -441.417,Z 979.783,A 0.000,B 0.000,C 90.000,E1 176.963} C_DIS
LIN {X -0.044,Y -452.593,Z 979.777,A 0.000,B 0.000,C 90.000,E1 175.812} C_DIS
LIN {X 0.044,Y -463.761,Z 979.770,A 0.000,B 0.000,C 90.000,E1 174.609} C_DIS
LIN {X 0.159,Y -471.741,Z 979.765,A 0.000,B 0.000,C 90.000,E1 173.685} C_DIS
LIN {X 0.021,Y -478.161,Z 979.761,A 0.000,B 0.000,C 90.000,E1 172.932} C_DIS
LIN {X 0.120,Y -486.678,Z 979.755,A 0.000,B 0.000,C 90.000,E1 171.837} C_DIS
LIN {X 0.170,Y -493.668,Z 979.750,A 0.000,B 0.000,C 90.000,E1 170.914} C_DIS
LIN {X 0.136,Y -501.453,Z 979.744,A 0.000,B 0.000,C 90.000,E1 169.859} C_DIS
LIN {X -0.218,Y -510.453,Z 979.736,A 0.000,B 0.000,C 90.000,E1 168.578} C_DIS
LIN {X 0.098,Y -519.087,Z 979.729,A 0.000,B 0.000,C 90.000,E1 167.229} C_DIS
LIN {X -0.096,Y -525.528,Z 979.723,A 0.000,B 0.000,C 90.000,E1 166.228} C_DIS
LIN {X 0.126,Y -532.625,Z 979.717,A 0.000,B 0.000,C 90.000,E1 165.046} C_DIS
LIN {X -0.225,Y -540.401,Z 979.710,A 0.000,B 0.000,C 90.000,E1 163.795} C_DIS
LIN {X 0.063,Y -547.745,Z 979.703,A 0.000,B 0.000,C 90.000,E1 162.489} C_DIS
LIN {X 0.011,Y -553.471,Z 979.697,A 0.000,B 0.000,C 90.000,E1 161.511} C_DIS
LIN {X 0.161,Y -562.730,Z 979.688,A 0.000,B 0.000,C 90.000,E1 159.826} C_DIS
LIN {X 0.207,Y -568.636,Z 979.682,A 0.000,B 0.000,C 90.000,E1 158.720} C_DIS
LIN {X -0.194,Y -574.235,Z 979.676,A 0.000,B 0.000,C 90.000,E1 157.667} C_DIS
LIN {X 0.238,Y -579.440,Z 979.670,A 0.000,B 0.000,C 90.000,E1 156.538} C_DIS
LIN {X -0.021,Y -584.346,Z 979.664,A 0.000,B 0.000,C 90.000,E1 155.485} C_DIS
LIN {X 0.135,Y -587.718,Z 979.659,A 0.000,B 0.000,C 90.000,E1 154.665} C_DIS
LIN {X -0.206,Y -590.890,Z 979.655,A 0.000,B 0.000,C 90.000,E1 153.896} C_DIS
LIN {X -0.085,Y -594.676,Z 979.649,A 0.000,B 0.000,C 90.000,E1 152.820} C_DIS
LIN {X -0.083,Y -597.281,Z 979.645,A 0.000,B 0.000,C 90.000,E1 152.025} C_DIS
LIN {X -0.121,Y -600.594,Z 979.639,A 0.000,B 0.000,C 90.000,E1 150.973} C_DIS
LIN {X -0.247,Y -605.393,Z 979.630,A 0.000,B 0.000,C 90.000,E1 149.410} C_DIS
LIN {X 0.339,Y -610.119,Z 979.621,A 0.000,B 0.000,C 90.000,E1 147.788} C_DIS
LIN {X 0.227,Y -614.015,Z 979.614,A 0.000,B 0.000,C 90.000,E1 146.501} C_DIS
LIN {X 0.213,Y -617.174,Z 979.608,A 0.000,B 0.000,C 90.000,E1 145.468} C_DIS
LIN {X -0.170,Y -622.575,Z 979.598,A 0.000,B 0.000,C 90.000,E1 143.703} C_DIS
LIN {X 0.135,Y -626.377,Z 979.591,A 0.000,B 0.000,C 90.000,E1 142.396} C_DIS
LIN {X 0.155,Y -629.496,Z 979.586,A 0.000,B 0.000,C 90.000,E1 141.376} C_DIS
LIN {X 0.050,Y -634.020,Z 979.577,A 0.000,B 0.000,C 90.000,E1 139.865} C_DIS
LIN {X -0.114,Y -638.356,Z 979.569,A 0.000,B 0.000,C 90.000,E1 138.366} C_DIS
LIN {X -0.294,Y -644.387,Z 979.558,A 0.000,B 0.000,C 90.000,E1 136.377} C_DIS
LIN {X 0.158,Y -649.894,Z 979.548,A 0.000,B 0.000,C 90.000,E1 134.595} C_DIS
LIN {X 0.219,Y -657.435,Z 979.536,A 0.000,B 0.000,C 90.000,E1 132.366} C_DIS
LIN {X 0.124,Y -664.581,Z 979.525,A 0.000,B 0.000,C 90.000,E1 130.415} C_DIS
LIN {X 0.141,Y -668.965,Z 979.518,A 0.000,B 0.000,C 90.000,E1 129.197} C_DIS
LIN {X 0.322,Y -673.901,Z 979.510,A 0.000,B 0.000,C 90.000,E1 127.729} C_DIS
LIN {X -0.363,Y -677.645,Z 979.503,A 0.000,B 0.000,C 90.000,E1 126.583} C_DIS
LIN {X 0.119,Y -681.978,Z 979.495,A 0.000,B 0.000,C 90.000,E1 125.105} C_DIS
LIN {X -0.082,Y -684.074,Z 979.491,A 0.000,B 0.000,C 90.000,E1 124.405} C_DIS
LIN {X -0.070,Y -686.697,Z 979.486,A 0.000,B 0.000,C 90.000,E1 123.452} C_DIS
LIN {X -0.163,Y -691.083,Z 979.477,A 0.000,B 0.000,C 90.000,E1 121.799} C_DIS
LIN {X -0.069,Y -693.388,Z 979.471,A 0.000,B 0.000,C 90.000,E1 120.846} C_DIS
LIN {X 0.053,Y -694.958,Z 979.467,A 0.000,B 0.000,C 90.000,E1 120.129} C_DIS
LIN {X 0.196,Y -696.391,Z 979.464,A 0.000,B 0.000,C 90.000,E1 119.411} C_DIS
LIN {X -0.256,Y -697.514,Z 979.460,A 0.000,B 0.000,C 90.000,E1 118.743} C_DIS
LIN {X -0.089,Y -698.351,Z 979.456,A 0.000,B 0.000,C 90.000,E1 118.025} C_DIS
LIN {X -0.054,Y -699.681,Z 979.448,A 0.000,B 0.000,C 90.000,E1 116.616} C_DIS
LIN {X -0.267,Y -700.560,Z 979.441,A 0.000,B 0.000,C 90.000,E1 115.463} C_DIS
LIN {X 0.254,Y -700.851,Z 979.438,A 0.000,B 0.000,C 90.000,E1 114.719} C_DIS
LIN {X 0.160,Y -700.911,Z 979.435,A 0.000,B 0.000,C 90.000,E1 114.259} C_DIS
LIN {X -0.224,Y -700.518,Z 979.432,A 0.000,B 0.000,C 90.000,E1 113.823} C_DIS
LIN {X 0.045,Y -700.220,Z 979.431,A 0.000,B 0.000,C 90.000,E1 113.567} C_DIS
LIN {X 0.301,Y -698.648,Z 979.428,A 0.000,B 0.000,C 90.000,E1 113.078} C_DIS
LIN {X -0.352,Y -697.560,Z 979.427,A 0.000,B 0.000,C 90.000,E1 112.898} C_DIS
LIN {X -0.091,Y -695.469,Z 979.426,A 0.000,B 0.000,C 90.000,E1 112.642} C_DIS
LIN {X 0.044,Y -691.887,Z 979.424,A 0.000,B 0.000,C 90.000,E1 112.280} C_DIS
LIN {X 0.193,Y -690.064,Z 979.423,A 0.000,B 0.000,C 90.000,E1 112.153} C_DIS
LIN {X 0.134,Y -685.264,Z 979.422,A 0.000,B 0.000,C 90.000,E1 111.972} C_DIS
LIN {X 0.120,Y -680.160,Z 979.421,A 0.000,B 0.000,C 90.000,E1 111.844} C_DIS
LIN {X 0.016,Y -676.178,Z 979.421,A 0.000,B 0.000,C 90.000,E1 111.770} C_DIS
LIN {X -0.225,Y -674.373,Z 979.421,A 0.000,B 0.000,C 90.000,E1 111.770} C_DIS
LIN {X 0.352,Y -669.232,Z 979.421,A 0.000,B 0.000,C 90.000,E1 111.716} C_DIS
LIN {X 0.284,Y -624.962,Z 979.421,A 0.000,B 0.000,C 90.000,E1 111.716} C_DIS
LIN {X -0.233,Y -622.085,Z 979.421,A 0.000,B 0.000,C 90.000,E1 111.716} C_DIS
LIN {X -0.202,Y -616.308,Z 979.420,A 0.000,B 0.000,C 90.000,E1 111.589} C_DIS
LIN {X 0.033,Y -609.379,Z 979.419,A 0.000,B 0.000,C 90.000,E1 111.354} C_DIS
LIN {X -0.009,Y -603.162,Z 979.417,A 0.000,B 0.000,C 90.000,E1 111.099} C_DIS
LIN {X -0.162,Y -597.100,Z 979.415,A 0.000,B 0.000,C 90.000,E1 110.791} C_DIS
LIN {X 0.003,Y -590.875,Z 979.413,A 0.000,B 0.000,C 90.000,E1 110.355} C_DIS
LIN {X -0.205,Y -578.871,Z 979.408,A 0.000,B 0.000,C 90.000,E1 109.450} C_DIS
LIN {X 0.060,Y -574.481,Z 979.406,A 0.000,B 0.000,C 90.000,E1 109.087} C_DIS
LIN {X -0.191,Y -566.109,Z 979.403,A 0.000,B 0.000,C 90.000,E1 108.598} C_DIS
LIN {X -0.105,Y -552.012,Z 979.399,A 0.000,B 0.000,C 90.000,E1 107.873} C_DIS
LIN {X 0.266,Y -549.730,Z 979.398,A 0.000,B 0.000,C 90.000,E1 107.638} C_DIS
LIN {X 0.228,Y -549.700,Z 979.398,A 0.000,B 0.000,C 90.000,E1 107.638} C_DIS
LIN {X 0.112,Y -549.391,Z 979.397,A 0.000,B 0.000,C 90.000,E1 107.511} C_DIS
LIN {X 0.205,Y -549.266,Z 979.396,A 0.000,B 0.000,C 90.000,E1 107.221} C_DIS
LIN {X -0.024,Y -550.223,Z 979.382,A 0.000,B 0.000,C 90.000,E1 104.717} C_DIS
LIN {X 0.044,Y -551.741,Z 979.368,A 0.000,B 0.000,C 90.000,E1 102.187} C_DIS
LIN {X 0.044,Y -554.068,Z 979.354,A 0.000,B 0.000,C 90.000,E1 99.670} C_DIS
LIN {X 0.030,Y -555.541,Z 979.346,A 0.000,B 0.000,C 90.000,E1 98.276} C_DIS
LIN {X 0.022,Y -557.163,Z 979.337,A 0.000,B 0.000,C 90.000,E1 96.606} C_DIS
LIN {X -0.015,Y -558.250,Z 979.329,A 0.000,B 0.000,C 90.000,E1 95.220} C_DIS
LIN {X -0.093,Y -559.187,Z 979.321,A 0.000,B 0.000,C 90.000,E1 93.841} C_DIS
LIN {X 0.280,Y -559.787,Z 979.315,A 0.000,B 0.000,C 90.000,E1 92.694} C_DIS
LIN {X 0.102,Y -560.410,Z 979.309,A 0.000,B 0.000,C 90.000,E1 91.604} C_DIS
LIN {X 0.013,Y -561.102,Z 979.301,A 0.000,B 0.000,C 90.000,E1 90.229} C_DIS
LIN {X -0.062,Y -561.599,Z 979.294,A 0.000,B 0.000,C 90.000,E1 88.854} C_DIS
LIN {X -0.021,Y -562.001,Z 979.284,A 0.000,B 0.000,C 90.000,E1 87.192} C_DIS
LIN {X -0.035,Y -562.243,Z 979.277,A 0.000,B 0.000,C 90.000,E1 85.812} C_DIS
LIN {X 0.194,Y -562.491,Z 979.266,A 0.000,B 0.000,C 90.000,E1 83.856} C_DIS
LIN {X 0.083,Y -562.864,Z 979.254,A 0.000,B 0.000,C 90.000,E1 81.659} C_DIS
LIN {X -0.097,Y -563.500,Z 979.243,A 0.000,B 0.000,C 90.000,E1 79.746} C_DIS
LIN {X 0.274,Y -564.656,Z 979.229,A 0.000,B 0.000,C 90.000,E1 77.229} C_DIS
LIN {X 0.089,Y -566.066,Z 979.217,A 0.000,B 0.000,C 90.000,E1 75.046} C_DIS
LIN {X -0.086,Y -567.393,Z 979.206,A 0.000,B 0.000,C 90.000,E1 73.142} C_DIS
LIN {X -0.025,Y -568.317,Z 979.199,A 0.000,B 0.000,C 90.000,E1 71.764} C_DIS
LIN {X 0.037,Y -569.362,Z 979.190,A 0.000,B 0.000,C 90.000,E1 70.115} C_DIS
LIN {X -0.222,Y -570.089,Z 979.182,A 0.000,B 0.000,C 90.000,E1 68.773} C_DIS
LIN {X -0.091,Y -570.600,Z 979.176,A 0.000,B 0.000,C 90.000,E1 67.667} C_DIS
LIN {X -0.301,Y -571.221,Z 979.167,A 0.000,B 0.000,C 90.000,E1 66.049} C_DIS
LIN {X -0.104,Y -571.658,Z 979.159,A 0.000,B 0.000,C 90.000,E1 64.665} C_DIS
LIN {X -0.163,Y -572.046,Z 979.152,A 0.000,B 0.000,C 90.000,E1 63.307} C_DIS
LIN {X 0.136,Y -572.373,Z 979.143,A 0.000,B 0.000,C 90.000,E1 61.641} C_DIS
LIN {X 0.203,Y -572.567,Z 979.133,A 0.000,B 0.000,C 90.000,E1 59.999} C_DIS
LIN {X -0.055,Y -572.723,Z 979.126,A 0.000,B 0.000,C 90.000,E1 58.663} C_DIS
LIN {X -0.004,Y -572.906,Z 979.118,A 0.000,B 0.000,C 90.000,E1 57.296} C_DIS
LIN {X -0.132,Y -572.967,Z 979.109,A 0.000,B 0.000,C 90.000,E1 55.674} C_DIS
LIN {X -0.042,Y -572.911,Z 979.105,A 0.000,B 0.000,C 90.000,E1 54.848} C_DIS
LIN {X 0.055,Y -572.582,Z 979.099,A 0.000,B 0.000,C 90.000,E1 53.749} C_DIS
LIN {X -0.181,Y -572.166,Z 979.093,A 0.000,B 0.000,C 90.000,E1 52.683} C_DIS
LIN {X -0.076,Y -571.577,Z 979.087,A 0.000,B 0.000,C 90.000,E1 51.582} C_DIS
LIN {X 0.330,Y -570.989,Z 979.082,A 0.000,B 0.000,C 90.000,E1 50.723} C_DIS
LIN {X -0.025,Y -570.010,Z 979.076,A 0.000,B 0.000,C 90.000,E1 49.666} C_DIS
LIN {X 0.036,Y -568.811,Z 979.070,A 0.000,B 0.000,C 90.000,E1 48.566} C_DIS
LIN {X 0.222,Y -568.159,Z 979.067,A 0.000,B 0.000,C 90.000,E1 48.000} C_DIS
LIN {X 0.205,Y -566.439,Z 979.061,A 0.000,B 0.000,C 90.000,E1 46.905} C_DIS
LIN {X -0.320,Y -564.989,Z 979.056,A 0.000,B 0.000,C 90.000,E1 46.134} C_DIS
LIN {X -0.067,Y -563.339,Z 979.052,A 0.000,B 0.000,C 90.000,E1 45.283} C_DIS
LIN {X -0.162,Y -560.854,Z 979.045,A 0.000,B 0.000,C 90.000,E1 44.190} C_DIS
LIN {X 0.099,Y -557.781,Z 979.039,A 0.000,B 0.000,C 90.000,E1 43.056} C_DIS
LIN {X -0.168,Y -556.107,Z 979.036,A 0.000,B 0.000,C 90.000,E1 42.528} C_DIS
LIN {X -0.008,Y -553.269,Z 979.032,A 0.000,B 0.000,C 90.000,E1 41.676} C_DIS
LIN {X -0.299,Y -551.184,Z 979.029,A 0.000,B 0.000,C 90.000,E1 41.148} C_DIS
LIN {X 0.172,Y -548.972,Z 979.025,A 0.000,B 0.000,C 90.000,E1 40.539} C_DIS
LIN {X -0.102,Y -545.320,Z 979.021,A 0.000,B 0.000,C 90.000,E1 39.725} C_DIS
LIN {X -0.078,Y -541.331,Z 979.016,A 0.000,B 0.000,C 90.000,E1 38.874} C_DIS
LIN {X -0.179,Y -536.182,Z 979.010,A 0.000,B 0.000,C 90.000,E1 37.890} C_DIS
LIN {X 0.143,Y -529.882,Z 979.004,A 0.000,B 0.000,C 90.000,E1 36.710} C_DIS
LIN {X -0.230,Y -524.895,Z 978.999,A 0.000,B 0.000,C 90.000,E1 35.884} C_DIS
LIN {X 0.031,Y -517.701,Z 978.993,A 0.000,B 0.000,C 90.000,E1 34.692} C_DIS
LIN {X -0.274,Y -512.762,Z 978.989,A 0.000,B 0.000,C 90.000,E1 33.992} C_DIS
LIN {X 0.173,Y -509.662,Z 978.986,A 0.000,B 0.000,C 90.000,E1 33.499} C_DIS
LIN {X 0.217,Y -504.179,Z 978.982,A 0.000,B 0.000,C 90.000,E1 32.752} C_DIS
LIN {X -0.089,Y -500.643,Z 978.980,A 0.000,B 0.000,C 90.000,E1 32.339} C_DIS
LIN {X 0.012,Y -496.904,Z 978.977,A 0.000,B 0.000,C 90.000,E1 31.878} C_DIS
LIN {X 0.218,Y -491.654,Z 978.974,A 0.000,B 0.000,C 90.000,E1 31.258} C_DIS
LIN {X -0.149,Y -486.190,Z 978.971,A 0.000,B 0.000,C 90.000,E1 30.718} C_DIS
LIN {X 0.146,Y -481.975,Z 978.968,A 0.000,B 0.000,C 90.000,E1 30.256} C_DIS
LIN {X 0.117,Y -471.935,Z 978.963,A 0.000,B 0.000,C 90.000,E1 29.283} C_DIS
LIN {X 0.038,Y -466.023,Z 978.960,A 0.000,B 0.000,C 90.000,E1 28.743} C_DIS
LIN {X -0.266,Y -455.651,Z 978.955,A 0.000,B 0.000,C 90.000,E1 27.847} C_DIS
LIN {X 0.183,Y -446.504,Z 978.950,A 0.000,B 0.000,C 90.000,E1 27.001} C_DIS
LIN {X 0.178,Y -421.142,Z 978.938,A 0.000,B 0.000,C 90.000,E1 24.771} C_DIS
LIN {X -0.160,Y -403.588,Z 978.928,A 0.000,B 0.000,C 90.000,E1 23.078} C_DIS
LIN {X 0.079,Y -398.421,Z 978.925,A 0.000,B 0.000,C 90.000,E1 22.461} C_DIS
LIN {X 0.049,Y -394.942,Z 978.922,A 0.000,B 0.000,C 90.000,E1 22.025} C_DIS
LIN {X -0.106,Y -392.211,Z 978.920,A 0.000,B 0.000,C 90.000,E1 21.589} C_DIS
LIN {X -0.028,Y -390.625,Z 978.917,A 0.000,B 0.000,C 90.000,E1 21.046} C_DIS
LIN {X 0.195,Y -389.937,Z 978.913,A 0.000,B 0.000,C 90.000,E1 20.301} C_DIS
LIN {X -0.110,Y -389.998,Z 978.910,A 0.000,B 0.000,C 90.000,E1 19.812} C_DIS
LIN {X -0.098,Y -395.220,Z 978.880,A 0.000,B 0.000,C 90.000,E1 14.481} C_DIS
LIN {X -0.024,Y -399.481,Z 978.863,A 0.000,B 0.000,C 90.000,E1 11.299} C_DIS
LIN {X -0.106,Y -404.099,Z 978.847,A 0.000,B 0.000,C 90.000,E1 8.511} C_DIS
LIN {X -0.145,Y -409.319,Z 978.832,A 0.000,B 0.000,C 90.000,E1 5.739} C_DIS
LIN {X -0.100,Y -415.102,Z 978.817,A 0.000,B 0.000,C 90.000,E1 2.980} C_DIS
LIN {X 0.028,Y -420.315,Z 978.804,A 0.000,B 0.000,C 90.000,E1 0.745} C_DIS
LIN {X 0.000,Y -423.050,Z 978.800,A 0.000,B 0.000,C 90.000,E1 360.000} C_DIS
LIN {X -0.162,Y -425.145,Z 978.798,A 0.000,B 0.000,C 90.000,E1 359.656} C_DIS
LIN {X -0.033,Y -427.479,Z 978.796,A 0.000,B 0.000,C 90.000,E1 359.312} C_DIS
LIN {X -0.005,Y -428.923,Z 978.795,A 0.000,B 0.000,C 90.000,E1 359.141} C_DIS
LIN {X 0.150,Y -433.504,Z 978.793,A 0.000,B 0.000,C 90.000,E1 358.740} C_DIS
LIN {X -0.178,Y -441.223,Z 978.791,A 0.000,B 0.000,C 90.000,E1 358.339} C_DIS
LIN {X 0.017,Y -456.470,Z 978.786,A 0.000,B 0.000,C 90.000,E1 357.478} C_DIS
LIN {X 0.088,Y -469.945,Z 978.782,A 0.000,B 0.000,C 90.000,E1 356.731} C_DIS
LIN {X -0.075,Y -481.671,Z 978.778,A 0.000,B 0.000,C 90.000,E1 356.102} C_DIS
LIN {X 0.205,Y -493.046,Z 978.775,A 0.000,B 0.000,C 90.000,E1 355.412} C_DIS
LIN {X -0.142,Y -504.407,Z 978.771,A 0.000,B 0.000,C 90.000,E1 354.780} C_DIS
LIN {X -0.106,Y -510.845,Z 978.769,A 0.000,B 0.000,C 90.000,E1 354.375} C_DIS
LIN {X 0.090,Y -520.016,Z 978.765,A 0.000,B 0.000,C 90.000,E1 353.742} C_DIS
LIN {X -0.153,Y -527.683,Z 978.762,A 0.000,B 0.000,C 90.000,E1 353.223} C_DIS
LIN {X -0.011,Y -532.076,Z 978.760,A 0.000,B 0.000,C 90.000,E1 352.875} C_DIS
LIN {X -0.130,Y -537.879,Z 978.758,A 0.000,B 0.000,C 90.000,E1 352.413} C_DIS
LIN {X 0.081,Y -543.537,Z 978.755,A 0.000,B 0.000,C 90.000,E1 351.894} C_DIS
LIN {X 0.150,Y -550.031,Z 978.752,A 0.000,B 0.000,C 90.000,E1 351.254} C_DIS
LIN {X 0.090,Y -555.059,Z 978.749,A 0.000,B 0.000,C 90.000,E1 350.735} C_DIS
LIN {X 0.146,Y -560.925,Z 978.745,A 0.000,B 0.000,C 90.000,E1 350.038} C_DIS
LIN {X 0.204,Y -566.247,Z 978.741,A 0.000,B 0.000,C 90.000,E1 349.342} C_DIS
LIN {X -0.253,Y -571.172,Z 978.737,A 0.000,B 0.000,C 90.000,E1 348.701} C_DIS
LIN {X 0.007,Y -575.566,Z 978.733,A 0.000,B 0.000,C 90.000,E1 347.993} C_DIS
LIN {X 0.187,Y -579.583,Z 978.730,A 0.000,B 0.000,C 90.000,E1 347.297} C_DIS
LIN {X 0.197,Y -584.906,Z 978.724,A 0.000,B 0.000,C 90.000,E1 346.353} C_DIS
LIN {X -0.064,Y -589.123,Z 978.720,A 0.000,B 0.000,C 90.000,E1 345.574} C_DIS
LIN {X 0.266,Y -595.712,Z 978.712,A 0.000,B 0.000,C 90.000,E1 344.212} C_DIS
LIN {X 0.182,Y -601.255,Z 978.706,A 0.000,B 0.000,C 90.000,E1 343.032} C_DIS
LIN {X 0.272,Y -604.787,Z 978.701,A 0.000,B 0.000,C 90.000,E1 342.236} C_DIS
LIN {X -0.125,Y -610.182,Z 978.694,A 0.000,B 0.000,C 90.000,E1 340.967} C_DIS
LIN {X -0.135,Y -613.249,Z 978.690,A 0.000,B 0.000,C 90.000,E1 340.188} C_DIS
LIN {X 0.057,Y -617.082,Z 978.684,A 0.000,B 0.000,C 90.000,E1 339.135} C_DIS
LIN {X 0.066,Y -621.467,Z 978.677,A 0.000,B 0.000,C 90.000,E1 337.847} C_DIS
LIN {X 0.136,Y -625.502,Z 978.670,A 0.000,B 0.000,C 90.000,E1 336.561} C_DIS
LIN {X -0.064,Y -629.264,Z 978.663,A 0.000,B 0.000,C 90.000,E1 335.305} C_DIS
LIN {X 0.007,Y -631.384,Z 978.659,A 0.000,B 0.000,C 90.000,E1 334.537} C_DIS
LIN {X 0.180,Y -634.489,Z 978.652,A 0.000,B 0.000,C 90.000,E1 333.256} C_DIS
LIN {X -0.206,Y -636.818,Z 978.646,A 0.000,B 0.000,C 90.000,E1 332.281} C_DIS
LIN {X 0.051,Y -639.477,Z 978.639,A 0.000,B 0.000,C 90.000,E1 331.001} C_DIS
LIN {X 0.037,Y -641.452,Z 978.633,A 0.000,B 0.000,C 90.000,E1 329.999} C_DIS
LIN {X 0.055,Y -643.340,Z 978.628,A 0.000,B 0.000,C 90.000,E1 328.997} C_DIS
LIN {X 0.098,Y -644.964,Z 978.622,A 0.000,B 0.000,C 90.000,E1 327.995} C_DIS
LIN {X 0.156,Y -646.417,Z 978.617,A 0.000,B 0.000,C 90.000,E1 326.993} C_DIS
LIN {X 0.104,Y -647.968,Z 978.610,A 0.000,B 0.000,C 90.000,E1 325.754} C_DIS
LIN {X 0.016,Y -648.974,Z 978.604,A 0.000,B 0.000,C 90.000,E1 324.769} C_DIS
LIN {X -0.093,Y -650.120,Z 978.596,A 0.000,B 0.000,C 90.000,E1 323.290} C_DIS
LIN {X -0.307,Y -651.036,Z 978.588,A 0.000,B 0.000,C 90.000,E1 321.823} C_DIS
LIN {X -0.022,Y -651.621,Z 978.581,A 0.000,B 0.000,C 90.000,E1 320.561} C_DIS
LIN {X -0.261,Y -652.378,Z 978.571,A 0.000,B 0.000,C 90.000,E1 318.852} C_DIS
LIN {X -0.201,Y -654.001,Z 978.558,A 0.000,B 0.000,C 90.000,E1 316.377} C_DIS
LIN {X 0.064,Y -654.978,Z 978.551,A 0.000,B 0.000,C 90.000,E1 315.121} C_DIS
LIN {X -0.243,Y -656.705,Z 978.538,A 0.000,B 0.000,C 90.000,E1 312.933} C_DIS
LIN {X 0.041,Y -657.909,Z 978.530,A 0.000,B 0.000,C 90.000,E1 311.434} C_DIS
LIN {X -0.068,Y -658.721,Z 978.523,A 0.000,B 0.000,C 90.000,E1 310.216} C_DIS
LIN {X -0.077,Y -659.514,Z 978.517,A 0.000,B 0.000,C 90.000,E1 308.991} C_DIS
LIN {X -0.100,Y -660.189,Z 978.508,A 0.000,B 0.000,C 90.000,E1 307.523} C_DIS
LIN {X -0.024,Y -660.578,Z 978.503,A 0.000,B 0.000,C 90.000,E1 306.537} C_DIS
LIN {X 0.048,Y -660.904,Z 978.494,A 0.000,B 0.000,C 90.000,E1 304.818} C_DIS
LIN {X 0.279,Y -661.317,Z 978.484,A 0.000,B 0.000,C 90.000,E1 303.086} C_DIS
LIN {X -0.027,Y -662.632,Z 978.470,A 0.000,B 0.000,C 90.000,E1 300.669} C_DIS
LIN {X 0.006,Y -668.766,Z 978.443,A 0.000,B 0.000,C 90.000,E1 295.796} C_DIS
LIN {X -0.069,Y -670.893,Z 978.437,A 0.000,B 0.000,C 90.000,E1 294.591} C_DIS
LIN {X -0.287,Y -672.476,Z 978.431,A 0.000,B 0.000,C 90.000,E1 293.643} C_DIS
LIN {X -0.044,Y -673.498,Z 978.427,A 0.000,B 0.000,C 90.000,E1 292.898} C_DIS
LIN {X 0.039,Y -673.946,Z 978.425,A 0.000,B 0.000,C 90.000,E1 292.408} C_DIS
LIN {X 0.381,Y -673.893,Z 978.422,A 0.000,B 0.000,C 90.000,E1 291.897} C_DIS
LIN {X -0.326,Y -673.767,Z 978.421,A 0.000,B 0.000,C 90.000,E1 291.716} C_DIS
LIN {X -0.238,Y -672.729,Z 978.418,A 0.000,B 0.000,C 90.000,E1 291.227} C_DIS
LIN {X -0.074,Y -672.005,Z 978.417,A 0.000,B 0.000,C 90.000,E1 290.972} C_DIS
LIN {X 0.006,Y -671.341,Z 978.416,A 0.000,B 0.000,C 90.000,E1 290.844} C_DIS
LIN {X -0.153,Y -670.346,Z 978.415,A 0.000,B 0.000,C 90.000,E1 290.737} C_DIS
LIN {X -0.033,Y -665.506,Z 978.413,A 0.000,B 0.000,C 90.000,E1 290.248} C_DIS
LIN {X -0.304,Y -660.556,Z 978.411,A 0.000,B 0.000,C 90.000,E1 289.939} C_DIS
LIN {X 0.229,Y -653.410,Z 978.408,A 0.000,B 0.000,C 90.000,E1 289.450} C_DIS
LIN {X 0.108,Y -650.293,Z 978.407,A 0.000,B 0.000,C 90.000,E1 289.214} C_DIS
LIN {X 0.069,Y -650.274,Z 978.407,A 0.000,B 0.000,C 90.000,E1 289.214} C_DIS
LIN {X 0.316,Y -650.099,Z 978.407,A 0.000,B 0.000,C 90.000,E1 289.141} C_DIS
LIN {X 0.277,Y -650.105,Z 978.407,A 0.000,B 0.000,C 90.000,E1 289.141} C_DIS
LIN {X -0.161,Y -651.124,Z 978.405,A 0.000,B 0.000,C 90.000,E1 288.833} C_DIS
LIN {X 0.354,Y -652.931,Z 978.403,A 0.000,B 0.000,C 90.000,E1 288.417} C_DIS
LIN {X 0.248,Y -658.873,Z 978.397,A 0.000,B 0.000,C 90.000,E1 287.457} C_DIS
LIN {X 0.127,Y -662.945,Z 978.393,A 0.000,B 0.000,C 90.000,E1 286.732} C_DIS
LIN {X -0.012,Y -665.971,Z 978.390,A 0.000,B 0.000,C 90.000,E1 286.134} C_DIS
LIN {X -0.182,Y -667.824,Z 978.387,A 0.000,B 0.000,C 90.000,E1 285.662} C_DIS
LIN {X -0.338,Y -669.375,Z 978.384,A 0.000,B 0.000,C 90.000,E1 285.190} C_DIS
LIN {X 0.168,Y -670.621,Z 978.382,A 0.000,B 0.000,C 90.000,E1 284.662} C_DIS
LIN {X 0.036,Y -671.625,Z 978.379,A 0.000,B 0.000,C 90.000,E1 284.189} C_DIS
LIN {X 0.008,Y -672.731,Z 978.375,A 0.000,B 0.000,C 90.000,E1 283.467} C_DIS
LIN {X -0.269,Y -673.278,Z 978.372,A 0.000,B 0.000,C 90.000,E1 283.008} C_DIS
LIN {X 0.273,Y -673.648,Z 978.370,A 0.000,B 0.000,C 90.000,E1 282.479} C_DIS
LIN {X 0.158,Y -673.860,Z 978.367,A 0.000,B 0.000,C 90.000,E1 282.007} C_DIS
LIN {X -0.019,Y -673.754,Z 978.363,A 0.000,B 0.000,C 90.000,E1 281.299} C_DIS
LIN {X -0.269,Y -673.509,Z 978.360,A 0.000,B 0.000,C 90.000,E1 280.838} C_DIS
LIN {X 0.269,Y -672.985,Z 978.357,A 0.000,B 0.000,C 90.000,E1 280.310} C_DIS
LIN {X 0.022,Y -672.257,Z 978.355,A 0.000,B 0.000,C 90.000,E1 279.849} C_DIS
LIN {X -0.116,Y -671.247,Z 978.352,A 0.000,B 0.000,C 90.000,E1 279.378} C_DIS
LIN {X 0.292,Y -669.906,Z 978.349,A 0.000,B 0.000,C 90.000,E1 278.859} C_DIS
LIN {X 0.213,Y -669.178,Z 978.348,A 0.000,B 0.000,C 90.000,E1 278.624} C_DIS
LIN {X -0.051,Y -667.438,Z 978.345,A 0.000,B 0.000,C 90.000,E1 278.163} C_DIS
LIN {X -0.323,Y -665.427,Z 978.343,A 0.000,B 0.000,C 90.000,E1 277.701} C_DIS
LIN {X 0.052,Y -662.969,Z 978.340,A 0.000,B 0.000,C 90.000,E1 277.182} C_DIS
LIN {X -0.249,Y -660.118,Z 978.337,A 0.000,B 0.000,C 90.000,E1 276.720} C_DIS
LIN {X 0.187,Y -657.713,Z 978.335,A 0.000,B 0.000,C 90.000,E1 276.315} C_DIS
LIN {X -0.148,Y -654.106,Z 978.333,A 0.000,B 0.000,C 90.000,E1 275.853} C_DIS
LIN {X 0.035,Y -649.066,Z 978.329,A 0.000,B 0.000,C 90.000,E1 275.220} C_DIS
LIN {X 0.288,Y -644.625,Z 978.326,A 0.000,B 0.000,C 90.000,E1 274.702} C_DIS
LIN {X -0.154,Y -639.815,Z 978.324,A 0.000,B 0.000,C 90.000,E1 274.245} C_DIS
LIN {X 0.218,Y -634.703,Z 978.321,A 0.000,B 0.000,C 90.000,E1 273.726} C_DIS
LIN {X 0.068,Y -629.302,Z 978.318,A 0.000,B 0.000,C 90.000,E1 273.269} C_DIS
LIN {X 0.153,Y -625.109,Z 978.316,A 0.000,B 0.000,C 90.000,E1 272.922} C_DIS
LIN {X -0.056,Y -617.758,Z 978.313,A 0.000,B 0.000,C 90.000,E1 272.407} C_DIS
LIN {X -0.152,Y -611.590,Z 978.311,A 0.000,B 0.000,C 90.000,E1 272.007} C_DIS
LIN {X -0.208,Y -603.388,Z 978.309,A 0.000,B 0.000,C 90.000,E1 271.547} C_DIS
LIN {X 0.093,Y -598.320,Z 978.307,A 0.000,B 0.000,C 90.000,E1 271.260} C_DIS
LIN {X -0.153,Y -591.173,Z 978.305,A 0.000,B 0.000,C 90.000,E1 270.974} C_DIS
LIN {X 0.049,Y -585.807,Z 978.304,A 0.000,B 0.000,C 90.000,E1 270.745} C_DIS
LIN {X -0.148,Y -579.863,Z 978.303,A 0.000,B 0.000,C 90.000,E1 270.573} C_DIS
LIN {X 0.258,Y -570.710,Z 978.302,A 0.000,B 0.000,C 90.000,E1 270.286} C_DIS
LIN {X 0.182,Y -564.965,Z 978.301,A 0.000,B 0.000,C 90.000,E1 270.172} C_DIS
LIN {X 0.017,Y -557.467,Z 978.301,A 0.000,B 0.000,C 90.000,E1 270.115} C_DIS
LIN {X -0.013,Y -546.358,Z 978.301,A 0.000,B 0.000,C 90.000,E1 270.115} C_DIS
LIN {X 0.159,Y -544.556,Z 978.300,A 0.000,B 0.000,C 90.000,E1 270.000} C_DIS
LIN {X 0.091,Y -542.885,Z 978.300,A 0.000,B 0.000,C 90.000,E1 269.943} C_DIS
LIN {X 0.036,Y -542.713,Z 978.300,A 0.000,B 0.000,C 90.000,E1 269.943} C_DIS
LIN {X -0.023,Y -541.477,Z 978.290,A 0.000,B 0.000,C 90.000,E1 268.224} C_DIS
LIN {X 0.149,Y -540.270,Z 978.281,A 0.000,B 0.000,C 90.000,E1 266.502} C_DIS
LIN {X -0.244,Y -539.292,Z 978.273,A 0.000,B 0.000,C 90.000,E1 265.122} C_DIS
LIN {X -0.118,Y -538.485,Z 978.266,A 0.000,B 0.000,C 90.000,E1 263.970} C_DIS
LIN {X 0.037,Y -536.906,Z 978.257,A 0.000,B 0.000,C 90.000,E1 262.243} C_DIS
LIN {X 0.243,Y -535.473,Z 978.249,A 0.000,B 0.000,C 90.000,E1 260.792} C_DIS
LIN {X -0.157,Y -534.309,Z 978.243,A 0.000,B 0.000,C 90.000,E1 259.690} C_DIS
LIN {X 0.185,Y -532.040,Z 978.232,A 0.000,B 0.000,C 90.000,E1 257.645} C_DIS
LIN {X -0.248,Y -531.431,Z 978.228,A 0.000,B 0.000,C 90.000,E1 257.117} C_DIS
LIN {X -0.037,Y -528.056,Z 978.212,A 0.000,B 0.000,C 90.000,E1 254.212} C_DIS
LIN {X 0.016,Y -525.897,Z 978.201,A 0.000,B 0.000,C 90.000,E1 252.181} C_DIS
LIN {X 0.009,Y -524.124,Z 978.193,A 0.000,B 0.000,C 90.000,E1 250.732} C_DIS
LIN {X 0.115,Y -521.815,Z 978.183,A 0.000,B 0.000,C 90.000,E1 248.975} C_DIS
LIN {X 0.060,Y -519.597,Z 978.174,A 0.000,B 0.000,C 90.000,E1 247.230} C_DIS
LIN {X 0.018,Y -518.353,Z 978.169,A 0.000,B 0.000,C 90.000,E1 246.357} C_DIS
LIN {X -0.242,Y -516.152,Z 978.161,A 0.000,B 0.000,C 90.000,E1 244.921} C_DIS
LIN {X 0.016,Y -513.391,Z 978.151,A 0.000,B 0.000,C 90.000,E1 243.127} C_DIS
LIN {X -0.230,Y -511.487,Z 978.144,A 0.000,B 0.000,C 90.000,E1 241.975} C_DIS
LIN {X -0.264,Y -509.563,Z 978.138,A 0.000,B 0.000,C 90.000,E1 240.795} C_DIS
LIN {X -0.001,Y -506.950,Z 978.129,A 0.000,B 0.000,C 90.000,E1 239.282} C_DIS
LIN {X 0.150,Y -504.607,Z 978.123,A 0.000,B 0.000,C 90.000,E1 238.074} C_DIS
LIN {X 0.141,Y -501.533,Z 978.115,A 0.000,B 0.000,C 90.000,E1 236.580} C_DIS
LIN {X 0.066,Y -498.802,Z 978.108,A 0.000,B 0.000,C 90.000,E1 235.388} C_DIS
LIN {X 0.084,Y -494.671,Z 978.098,A 0.000,B 0.000,C 90.000,E1 233.577} C_DIS
LIN {X 0.201,Y -490.399,Z 978.088,A 0.000,B 0.000,C 90.000,E1 231.743} C_DIS
LIN {X -0.271,Y -488.293,Z 978.083,A 0.000,B 0.000,C 90.000,E1 230.884} C_DIS
LIN {X 0.194,Y -484.693,Z 978.074,A 0.000,B 0.000,C 90.000,E1 229.299} C_DIS
LIN {X 0.156,Y -479.760,Z 978.062,A 0.000,B 0.000,C 90.000,E1 227.148} C_DIS
LIN {X -0.253,Y -476.420,Z 978.053,A 0.000,B 0.000,C 90.000,E1 225.648} C_DIS
LIN {X 0.277,Y -473.024,Z 978.045,A 0.000,B 0.000,C 90.000,E1 224.028} C_DIS
LIN {X 0.172,Y -468.876,Z 978.034,A 0.000,B 0.000,C 90.000,E1 222.162} C_DIS
LIN {X 0.084,Y -466.881,Z 978.029,A 0.000,B 0.000,C 90.000,E1 221.229} C_DIS
LIN {X -0.116,Y -462.615,Z 978.019,A 0.000,B 0.000,C 90.000,E1 219.358} C_DIS
LIN {X 0.046,Y -457.579,Z 978.006,A 0.000,B 0.000,C 90.000,E1 217.111} C_DIS
LIN {X 0.074,Y -453.342,Z 977.996,A 0.000,B 0.000,C 90.000,E1 215.185} C_DIS
LIN {X 0.112,Y -449.128,Z 977.985,A 0.000,B 0.000,C 90.000,E1 213.245} C_DIS
LIN {X -0.132,Y -444.260,Z 977.972,A 0.000,B 0.000,C 90.000,E1 211.003} C_DIS
LIN {X 0.147,Y -440.741,Z 977.963,A 0.000,B 0.000,C 90.000,E1 209.333} C_DIS
LIN {X -0.022,Y -435.598,Z 977.950,A 0.000,B 0.000,C 90.000,E1 207.052} C_DIS
LIN {X 0.029,Y -433.497,Z 977.945,A 0.000,B 0.000,C 90.000,E1 206.052} C_DIS
LIN {X 0.062,Y -430.403,Z 977.937,A 0.000,B 0.000,C 90.000,E1 204.719} C_DIS
LIN {X 0.188,Y -424.296,Z 977.923,A 0.000,B 0.000,C 90.000,E1 202.025} C_DIS
LIN {X 0.240,Y -419.915,Z 977.911,A 0.000,B 0.000,C 90.000,E1 199.993} C_DIS
LIN {X 0.207,Y -414.368,Z 977.896,A 0.000,B 0.000,C 90.000,E1 197.275} C_DIS
LIN {X 0.016,Y -410.550,Z 977.885,A 0.000,B 0.000,C 90.000,E1 195.245} C_DIS
LIN {X -0.087,Y -407.375,Z 977.875,A 0.000,B 0.000,C 90.000,E1 193.536} C_DIS
LIN {X 0.142,Y -404.134,Z 977.866,A 0.000,B 0.000,C 90.000,E1 191.771} C_DIS
LIN {X 0.207,Y -400.198,Z 977.854,A 0.000,B 0.000,C 90.000,E1 189.670} C_DIS
LIN {X -0.164,Y -393.522,Z 977.832,A 0.000,B 0.000,C 90.000,E1 185.853} C_DIS
LIN {X 0.053,Y -392.497,Z 977.827,A 0.000,B 0.000,C 90.000,E1 184.759} C_DIS
LIN {X -0.112,Y -392.002,Z 977.823,A 0.000,B 0.000,C 90.000,E1 184.073} C_DIS
LIN {X -0.167,Y -391.959,Z 977.821,A 0.000,B 0.000,C 90.000,E1 183.726} C_DIS
LIN {X 0.143,Y -392.101,Z 977.819,A 0.000,B 0.000,C 90.000,E1 183.326} C_DIS
LIN {X 0.002,Y -393.042,Z 977.815,A 0.000,B 0.000,C 90.000,E1 182.636} C_DIS
LIN {X -0.130,Y -394.795,Z 977.811,A 0.000,B 0.000,C 90.000,E1 181.949} C_DIS
LIN {X 0.174,Y -397.028,Z 977.808,A 0.000,B 0.000,C 90.000,E1 181.375} C_DIS
LIN {X 0.198,Y -400.656,Z 977.804,A 0.000,B 0.000,C 90.000,E1 180.745} C_DIS
LIN {X -0.181,Y -406.130,Z 977.801,A 0.000,B 0.000,C 90.000,E1 180.115} C_DIS
LIN {X -0.003,Y -416.579,Z 977.795,A 0.000,B 0.000,C 90.000,E1 179.026} C_DIS
LIN {X 0.041,Y -428.629,Z 977.788,A 0.000,B 0.000,C 90.000,E1 177.879} C_DIS
LIN {X -0.074,Y -440.026,Z 977.782,A 0.000,B 0.000,C 90.000,E1 176.788} C_DIS
LIN {X -0.125,Y -449.803,Z 977.777,A 0.000,B 0.000,C 90.000,E1 175.812} C_DIS
LIN {X -0.157,Y -462.459,Z 977.769,A 0.000,B 0.000,C 90.000,E1 174.489} C_DIS
LIN {X -0.139,Y -471.600,Z 977.764,A 0.000,B 0.000,C 90.000,E1 173.451} C_DIS
LIN {X -0.182,Y -479.300,Z 977.758,A 0.000,B 0.000,C 90.000,E1 172.527} C_DIS
LIN {X 0.059,Y -485.533,Z 977.754,A 0.000,B 0.000,C 90.000,E1 171.724} C_DIS
LIN {X 0.136,Y -494.779,Z 977.747,A 0.000,B 0.000,C 90.000,E1 170.500} C_DIS
LIN {X -0.219,Y -501.404,Z 977.742,A 0.000,B 0.000,C 90.000,E1 169.634} C_DIS
LIN {X 0.026,Y -509.596,Z 977.736,A 0.000,B 0.000,C 90.000,E1 168.409} C_DIS
LIN {X 0.180,Y -520.325,Z 977.727,A 0.000,B 0.000,C 90.000,E1 166.769} C_DIS
LIN {X -0.204,Y -525.728,Z 977.722,A 0.000,B 0.000,C 90.000,E1 165.936} C_DIS
LIN {X -0.189,Y -532.024,Z 977.716,A 0.000,B 0.000,C 90.000,E1 164.921} C_DIS
LIN {X -0.028,Y -539.754,Z 977.709,A 0.000,B 0.000,C 90.000,E1 163.614} C_DIS
LIN {X -0.130,Y -546.386,Z 977.703,A 0.000,B 0.000,C 90.000,E1 162.489} C_DIS
LIN {X 0.196,Y -552.851,Z 977.696,A 0.000,B 0.000,C 90.000,E1 161.329} C_DIS
LIN {X 0.221,Y -560.734,Z 977.689,A 0.000,B 0.000,C 90.000,E1 159.934} C_DIS
LIN {X -0.083,Y -565.232,Z 977.684,A 0.000,B 0.000,C 90.000,E1 159.135} C_DIS
LIN {X -0.086,Y -571.651,Z 977.677,A 0.000,B 0.000,C 90.000,E1 157.901} C_DIS
LIN {X 0.168,Y -576.388,Z 977.672,A 0.000,B 0.000,C 90.000,E1 156.922} C_DIS
LIN {X 0.317,Y -579.566,Z 977.668,A 0.000,B 0.000,C 90.000,E1 156.230} C_DIS
LIN {X -0.341,Y -583.320,Z 977.664,A 0.000,B 0.000,C 90.000,E1 155.485} C_DIS
LIN {X -0.198,Y -586.732,Z 977.659,A 0.000,B 0.000,C 90.000,E1 154.665} C_DIS
LIN {X -0.022,Y -589.958,Z 977.655,A 0.000,B 0.000,C 90.000,E1 153.845} C_DIS
LIN {X -0.174,Y -593.828,Z 977.649,A 0.000,B 0.000,C 90.000,E1 152.794} C_DIS
LIN {X 0.073,Y -596.485,Z 977.644,A 0.000,B 0.000,C 90.000,E1 151.975} C_DIS
LIN {X -0.061,Y -600.588,Z 977.637,A 0.000,B 0.000,C 90.000,E1 150.667} C_DIS
LIN {X 0.110,Y -605.437,Z 977.628,A 0.000,B 0.000,C 90.000,E1 149.076} C_DIS
LIN {X -0.084,Y -609.389,Z 977.621,A 0.000,B 0.000,C 90.000,E1 147.788} C_DIS
LIN {X -0.158,Y -612.598,Z 977.615,A 0.000,B 0.000,C 90.000,E1 146.755} C_DIS
LIN {X -0.235,Y -616.526,Z 977.608,A 0.000,B 0.000,C 90.000,E1 145.468} C_DIS
LIN {X -0.091,Y -621.238,Z 977.599,A 0.000,B 0.000,C 90.000,E1 143.909} C_DIS
LIN {X -0.187,Y -625.087,Z 977.592,A 0.000,B 0.000,C 90.000,E1 142.637} C_DIS
LIN {X 0.157,Y -628.970,Z 977.585,A 0.000,B 0.000,C 90.000,E1 141.331} C_DIS
LIN {X 0.077,Y -632.792,Z 977.578,A 0.000,B 0.000,C 90.000,E1 140.070} C_DIS
LIN {X -0.051,Y -637.206,Z 977.570,A 0.000,B 0.000,C 90.000,E1 138.566} C_DIS
LIN {X 0.163,Y -643.294,Z 977.559,A 0.000,B 0.000,C 90.000,E1 136.539} C_DIS
LIN {X -0.263,Y -647.994,Z 977.550,A 0.000,B 0.000,C 90.000,E1 135.081} C_DIS
LIN {X -0.299,Y -656.370,Z 977.537,A 0.000,B 0.000,C 90.000,E1 132.609} C_DIS
LIN {X -0.013,Y -664.431,Z 977.524,A 0.000,B 0.000,C 90.000,E1 130.378} C_DIS
LIN {X 0.003,Y -667.967,Z 977.519,A 0.000,B 0.000,C 90.000,E1 129.402} C_DIS
LIN {X -0.259,Y -673.790,Z 977.510,A 0.000,B 0.000,C 90.000,E1 127.729} C_DIS
LIN {X -0.002,Y -677.565,Z 977.503,A 0.000,B 0.000,C 90.000,E1 126.503} C_DIS
LIN {X -0.080,Y -681.928,Z 977.495,A 0.000,B 0.000,C 90.000,E1 125.072} C_DIS
LIN {X 0.275,Y -684.035,Z 977.491,A 0.000,B 0.000,C 90.000,E1 124.326} C_DIS
LIN {X -0.087,Y -687.322,Z 977.484,A 0.000,B 0.000,C 90.000,E1 123.166} C_DIS
LIN {X -0.176,Y -691.056,Z 977.476,A 0.000,B 0.000,C 90.000,E1 121.750} C_DIS
LIN {X -0.075,Y -693.348,Z 977.471,A 0.000,B 0.000,C 90.000,E1 120.797} C_DIS
LIN {X 0.051,Y -694.900,Z 977.467,A 0.000,B 0.000,C 90.000,E1 120.079} C_DIS
LIN {X -0.410,Y -696.294,Z 977.463,A 0.000,B 0.000,C 90.000,E1 119.411} C_DIS
LIN {X 0.009,Y -697.725,Z 977.458,A 0.000,B 0.000,C 90.000,E1 118.437} C_DIS
LIN {X -0.172,Y -698.647,Z 977.453,A 0.000,B 0.000,C 90.000,E1 117.513} C_DIS
LIN {X -0.042,Y -699.555,Z 977.448,A 0.000,B 0.000,C 90.000,E1 116.565} C_DIS
LIN {X -0.251,Y -700.401,Z 977.441,A 0.000,B 0.000,C 90.000,E1 115.412} C_DIS
LIN {X -0.072,Y -700.656,Z 977.437,A 0.000,B 0.000,C 90.000,E1 114.695} C_DIS
LIN {X 0.180,Y -700.694,Z 977.435,A 0.000,B 0.000,C 90.000,E1 114.207} C_DIS
LIN {X -0.203,Y -700.268,Z 977.432,A 0.000,B 0.000,C 90.000,E1 113.770} C_DIS
LIN {X 0.066,Y -699.842,Z 977.431,A 0.000,B 0.000,C 90.000,E1 113.515} C_DIS
LIN {X -0.320,Y -698.307,Z 977.428,A 0.000,B 0.000,C 90.000,E1 113.078} C_DIS
LIN {X -0.189,Y -697.794,Z 977.427,A 0.000,B 0.000,C 90.000,E1 112.950} C_DIS
LIN {X -0.059,Y -696.992,Z 977.427,A 0.000,B 0.000,C 90.000,E1 112.823} C_DIS
LIN {X 0.176,Y -692.521,Z 977.424,A 0.000,B 0.000,C 90.000,E1 112.333} C_DIS
LIN {X 0.297,Y -691.061,Z 977.424,A 0.000,B 0.000,C 90.000,E1 112.206} C_DIS
LIN {X 0.158,Y -688.583,Z 977.423,A 0.000,B 0.000,C 90.000,E1 112.099} C_DIS
LIN {X -0.135,Y -684.533,Z 977.422,A 0.000,B 0.000,C 90.000,E1 111.972} C_DIS
LIN {X 0.283,Y -677.534,Z 977.421,A 0.000,B 0.000,C 90.000,E1 111.770} C_DIS
LIN {X 0.341,Y -674.752,Z 977.421,A 0.000,B 0.000,C 90.000,E1 111.716} C_DIS
LIN {X 0.288,Y -670.950,Z 977.421,A 0.000,B 0.000,C 90.000,E1 111.716} C_DIS
LIN {X 0.209,Y -625.668,Z 977.421,A 0.000,B 0.000,C 90.000,E1 111.716} C_DIS
LIN {X 0.196,Y -622.217,Z 977.420,A 0.000,B 0.000,C 90.000,E1 111.663} C_DIS
LIN {X 0.221,Y -616.495,Z 977.420,A 0.000,B 0.000,C 90.000,E1 111.535} C_DIS
LIN {X -0.131,Y -609.466,Z 977.419,A 0.000,B 0.000,C 90.000,E1 111.354} C_DIS
LIN {X -0.214,Y -603.232,Z 977.417,A 0.000,B 0.000,C 90.000,E1 111.099} C_DIS
LIN {X 0.175,Y -597.138,Z 977.415,A 0.000,B 0.000,C 90.000,E1 110.737} C_DIS
LIN {X 0.218,Y -589.982,Z 977.413,A 0.000,B 0.000,C 90.000,E1 110.248} C_DIS
LIN {X 0.038,Y -577.068,Z 977.407,A 0.000,B 0.000,C 90.000,E1 109.268} C_DIS
LIN {X 0.175,Y -574.121,Z 977.406,A 0.000,B 0.000,C 90.000,E1 109.033} C_DIS
LIN {X -0.211,Y -567.634,Z 977.404,A 0.000,B 0.000,C 90.000,E1 108.671} C_DIS
LIN {X 0.234,Y -559.102,Z 977.401,A 0.000,B 0.000,C 90.000,E1 108.181} C_DIS
LIN {X -0.042,Y -552.449,Z 977.399,A 0.000,B 0.000,C 90.000,E1 107.873} C_DIS
LIN {X 0.123,Y -549.806,Z 977.398,A 0.000,B 0.000,C 90.000,E1 107.638} C_DIS
LIN {X 0.086,Y -549.793,Z 977.398,A 0.000,B 0.000,C 90.000,E1 107.638} C_DIS
LIN {X -0.027,Y -549.356,Z 977.397,A 0.000,B 0.000,C 90.000,E1 107.457} C_DIS
LIN {X -0.107,Y -549.486,Z 977.392,A 0.000,B 0.000,C 90.000,E1 106.622} C_DIS
LIN {X 0.094,Y -550.480,Z 977.380,A 0.000,B 0.000,C 90.000,E1 104.356} C_DIS
LIN {X 0.157,Y -552.071,Z 977.366,A 0.000,B 0.000,C 90.000,E1 101.827} C_DIS
LIN {X -0.068,Y -554.200,Z 977.353,A 0.000,B 0.000,C 90.000,E1 99.613} C_DIS
LIN {X -0.078,Y -555.660,Z 977.346,A 0.000,B 0.000,C 90.000,E1 98.219} C_DIS
LIN {X -0.081,Y -557.261,Z 977.336,A 0.000,B 0.000,C 90.000,E1 96.549} C_DIS
LIN {X -0.115,Y -558.331,Z 977.329,A 0.000,B 0.000,C 90.000,E1 95.163} C_DIS
LIN {X -0.192,Y -559.256,Z 977.321,A 0.000,B 0.000,C 90.000,E1 93.784} C_DIS
LIN {X 0.096,Y -559.701,Z 977.316,A 0.000,B 0.000,C 90.000,E1 92.922} C_DIS
LIN {X -0.103,Y -560.341,Z 977.310,A 0.000,B 0.000,C 90.000,E1 91.835} C_DIS
LIN {X -0.081,Y -561.162,Z 977.301,A 0.000,B 0.000,C 90.000,E1 90.172} C_DIS
LIN {X -0.156,Y -561.612,Z 977.293,A 0.000,B 0.000,C 90.000,E1 88.797} C_DIS
LIN {X -0.115,Y -562.030,Z 977.284,A 0.000,B 0.000,C 90.000,E1 87.135} C_DIS
LIN {X -0.129,Y -562.281,Z 977.276,A 0.000,B 0.000,C 90.000,E1 85.755} C_DIS
LIN {X 0.099,Y -562.526,Z 977.266,A 0.000,B 0.000,C 90.000,E1 83.799} C_DIS
LIN {X 0.058,Y -562.946,Z 977.252,A 0.000,B 0.000,C 90.000,E1 81.319} C_DIS
LIN {X -0.196,Y -563.557,Z 977.243,A 0.000,B 0.000,C 90.000,E1 79.690} C_DIS
LIN {X 0.169,Y -564.691,Z 977.229,A 0.000,B 0.000,C 90.000,E1 77.173} C_DIS
LIN {X -0.019,Y -566.120,Z 977.217,A 0.000,B 0.000,C 90.000,E1 74.991} C_DIS
LIN {X 0.184,Y -567.264,Z 977.208,A 0.000,B 0.000,C 90.000,E1 73.323} C_DIS
LIN {X 0.242,Y -568.204,Z 977.200,A 0.000,B 0.000,C 90.000,E1 71.945} C_DIS
LIN {X -0.083,Y -569.396,Z 977.189,A 0.000,B 0.000,C 90.000,E1 70.061} C_DIS
LIN {X -0.347,Y -570.118,Z 977.182,A 0.000,B 0.000,C 90.000,E1 68.720} C_DIS
LIN {X -0.001,Y -570.591,Z 977.176,A 0.000,B 0.000,C 90.000,E1 67.592} C_DIS
LIN {X -0.035,Y -571.114,Z 977.168,A 0.000,B 0.000,C 90.000,E1 66.230} C_DIS
LIN {X 0.000,Y -571.626,Z 977.159,A 0.000,B 0.000,C 90.000,E1 64.588} C_DIS
LIN {X -0.310,Y -572.002,Z 977.151,A 0.000,B 0.000,C 90.000,E1 63.256} C_DIS
LIN {X 0.146,Y -572.266,Z 977.144,A 0.000,B 0.000,C 90.000,E1 61.847} C_DIS
LIN {X 0.205,Y -572.454,Z 977.135,A 0.000,B 0.000,C 90.000,E1 60.205} C_DIS
LIN {X -0.058,Y -572.603,Z 977.127,A 0.000,B 0.000,C 90.000,E1 58.869} C_DIS
LIN {X -0.188,Y -572.806,Z 977.118,A 0.000,B 0.000,C 90.000,E1 57.248} C_DIS
LIN {X -0.003,Y -572.831,Z 977.109,A 0.000,B 0.000,C 90.000,E1 55.595} C_DIS
LIN {X 0.087,Y -572.747,Z 977.104,A 0.000,B 0.000,C 90.000,E1 54.769} C_DIS
LIN {X -0.154,Y -572.401,Z 977.098,A 0.000,B 0.000,C 90.000,E1 53.703} C_DIS
LIN {X 0.264,Y -572.072,Z 977.094,A 0.000,B 0.000,C 90.000,E1 52.844} C_DIS
LIN {X -0.303,Y -571.342,Z 977.086,A 0.000,B 0.000,C 90.000,E1 51.537} C_DIS
LIN {X 0.095,Y -570.735,Z 977.082,A 0.000,B 0.000,C 90.000,E1 50.678} C_DIS
LIN {X 0.100,Y -569.702,Z 977.076,A 0.000,B 0.000,C 90.000,E1 49.585} C_DIS
LIN {X 0.156,Y -568.470,Z 977.070,A 0.000,B 0.000,C 90.000,E1 48.485} C_DIS
LIN {X 0.032,Y -567.356,Z 977.065,A 0.000,B 0.000,C 90.000,E1 47.676} C_DIS
LIN {X 0.008,Y -565.595,Z 977.059,A 0.000,B 0.000,C 90.000,E1 46.581} C_DIS
LIN {X 0.272,Y -564.045,Z 977.054,A 0.000,B 0.000,C 90.000,E1 45.729} C_DIS
LIN {X 0.113,Y -562.283,Z 977.050,A 0.000,B 0.000,C 90.000,E1 44.919} C_DIS
LIN {X -0.064,Y -560.261,Z 977.045,A 0.000,B 0.000,C 90.000,E1 44.109} C_DIS
LIN {X 0.141,Y -557.955,Z 977.040,A 0.000,B 0.000,C 90.000,E1 43.257} C_DIS
LIN {X 0.256,Y -556.327,Z 977.037,A 0.000,B 0.000,C 90.000,E1 42.690} C_DIS
LIN {X -0.018,Y -554.538,Z 977.034,A 0.000,B 0.000,C 90.000,E1 42.162} C_DIS
LIN {X 0.127,Y -551.478,Z 977.030,A 0.000,B 0.000,C 90.000,E1 41.310} C_DIS
LIN {X 0.234,Y -548.111,Z 977.025,A 0.000,B 0.000,C 90.000,E1 40.458} C_DIS
LIN {X -0.091,Y -545.685,Z 977.022,A 0.000,B 0.000,C 90.000,E1 39.930} C_DIS
LIN {X -0.018,Y -543.069,Z 977.019,A 0.000,B 0.000,C 90.000,E1 39.358} C_DIS
LIN {X 0.043,Y -540.288,Z 977.016,A 0.000,B 0.000,C 90.000,E1 38.785} C_DIS
LIN {X -0.155,Y -535.085,Z 977.010,A 0.000,B 0.000,C 90.000,E1 37.810} C_DIS
LIN {X -0.168,Y -528.670,Z 977.004,A 0.000,B 0.000,C 90.000,E1 36.664} C_DIS
LIN {X -0.240,Y -523.568,Z 976.999,A 0.000,B 0.000,C 90.000,E1 35.804} C_DIS
LIN {X 0.176,Y -517.220,Z 976.993,A 0.000,B 0.000,C 90.000,E1 34.739} C_DIS
LIN {X -0.245,Y -513.306,Z 976.990,A 0.000,B 0.000,C 90.000,E1 34.199} C_DIS
LIN {X 0.023,Y -509.142,Z 976.987,A 0.000,B 0.000,C 90.000,E1 33.579} C_DIS
LIN {X 0.063,Y -503.619,Z 976.982,A 0.000,B 0.000,C 90.000,E1 32.832} C_DIS
LIN {X -0.242,Y -500.037,Z 976.980,A 0.000,B 0.000,C 90.000,E1 32.418} C_DIS
LIN {X -0.282,Y -493.636,Z 976.976,A 0.000,B 0.000,C 90.000,E1 31.671} C_DIS
LIN {X 0.160,Y -486.820,Z 976.972,A 0.000,B 0.000,C 90.000,E1 30.875} C_DIS
LIN {X -0.119,Y -481.089,Z 976.969,A 0.000,B 0.000,C 90.000,E1 30.335} C_DIS
LIN {X 0.075,Y -471.324,Z 976.963,A 0.000,B 0.000,C 90.000,E1 29.361} C_DIS
LIN {X 0.015,Y -465.392,Z 976.960,A 0.000,B 0.000,C 90.000,E1 28.821} C_DIS
LIN {X -0.028,Y -456.530,Z 976.956,A 0.000,B 0.000,C 90.000,E1 28.025} C_DIS
LIN {X -0.239,Y -447.322,Z 976.951,A 0.000,B 0.000,C 90.000,E1 27.257} C_DIS
LIN {X -0.221,Y -423.233,Z 976.940,A 0.000,B 0.000,C 90.000,E1 25.155} C_DIS
LIN {X 0.129,Y -405.568,Z 976.930,A 0.000,B 0.000,C 90.000,E1 23.387} C_DIS
LIN {X -0.020,Y -397.589,Z 976.925,A 0.000,B 0.000,C 90.000,E1 22.514} C_DIS
LIN {X 0.154,Y -395.034,Z 976.923,A 0.000,B 0.000,C 90.000,E1 22.153} C_DIS
LIN {X -0.158,Y -393.883,Z 976.922,A 0.000,B 0.000,C 90.000,E1 22.025} C_DIS
LIN {X 0.057,Y -392.317,Z 976.921,A 0.000,B 0.000,C 90.000,E1 21.716} C_DIS
LIN {X -0.129,Y -391.616,Z 976.920,A 0.000,B 0.000,C 90.000,E1 21.589} C_DIS
LIN {X 0.094,Y -390.339,Z 976.917,A 0.000,B 0.000,C 90.000,E1 21.046} C_DIS
LIN {X -0.048,Y -389.876,Z 976.913,A 0.000,B 0.000,C 90.000,E1 20.355} C_DIS
LIN {X 0.071,Y -390.352,Z 976.907,A 0.000,B 0.000,C 90.000,E1 19.268} C_DIS
LIN {X 0.001,Y -395.068,Z 976.882,A 0.000,B 0.000,C 90.000,E1 14.662} C_DIS
LIN {X 0.076,Y -399.292,Z 976.864,A 0.000,B 0.000,C 90.000,E1 11.478} C_DIS
LIN {X 0.069,Y -402.620,Z 976.852,A 0.000,B 0.000,C 90.000,E1 9.378} C_DIS
LIN {X 0.011,Y -406.390,Z 976.841,A 0.000,B 0.000,C 90.000,E1 7.296} C_DIS
LIN {X -0.020,Y -411.120,Z 976.827,A 0.000,B 0.000,C 90.000,E1 4.878} C_DIS
LIN {X 0.045,Y -415.518,Z 976.816,A 0.000,B 0.000,C 90.000,E1 2.808} C_DIS
LIN {X 0.173,Y -420.328,Z 976.804,A 0.000,B 0.000,C 90.000,E1 0.745} C_DIS
LIN {X -0.182,Y -422.551,Z 976.801,A 0.000,B 0.000,C 90.000,E1 0.115} C_DIS
LIN {X 0.184,Y -424.961,Z 976.798,A 0.000,B 0.000,C 90.000,E1 359.599} C_DIS
LIN {X 0.208,Y -425.992,Z 976.797,A 0.000,B 0.000,C 90.000,E1 359.427} C_DIS
LIN {X -0.166,Y -428.660,Z 976.795,A 0.000,B 0.000,C 90.000,E1 359.141} C_DIS
LIN {X -0.093,Y -432.351,Z 976.793,A 0.000,B 0.000,C 90.000,E1 358.797} C_DIS
LIN {X -0.180,Y -433.896,Z 976.793,A 0.000,B 0.000,C 90.000,E1 358.682} C_DIS
LIN {X 0.027,Y -455.176,Z 976.786,A 0.000,B 0.000,C 90.000,E1 357.478} C_DIS
LIN {X -0.188,Y -470.338,Z 976.781,A 0.000,B 0.000,C 90.000,E1 356.674} C_DIS
LIN {X -0.198,Y -478.731,Z 976.779,A 0.000,B 0.000,C 90.000,E1 356.216} C_DIS
LIN {X -0.232,Y -491.799,Z 976.775,A 0.000,B 0.000,C 90.000,E1 355.469} C_DIS
LIN {X 0.086,Y -502.948,Z 976.771,A 0.000,B 0.000,C 90.000,E1 354.780} C_DIS
LIN {X -0.129,Y -510.855,Z 976.768,A 0.000,B 0.000,C 90.000,E1 354.318} C_DIS
LIN {X 0.068,Y -520.041,Z 976.765,A 0.000,B 0.000,C 90.000,E1 353.685} C_DIS
LIN {X -0.121,Y -527.677,Z 976.762,A 0.000,B 0.000,C 90.000,E1 353.166} C_DIS
LIN {X -0.031,Y -533.547,Z 976.760,A 0.000,B 0.000,C 90.000,E1 352.704} C_DIS
LIN {X 0.036,Y -539.063,Z 976.757,A 0.000,B 0.000,C 90.000,E1 352.243} C_DIS
LIN {X -0.177,Y -543.285,Z 976.755,A 0.000,B 0.000,C 90.000,E1 351.894} C_DIS
LIN {X -0.089,Y -549.791,Z 976.751,A 0.000,B 0.000,C 90.000,E1 351.254} C_DIS
LIN {X -0.141,Y -554.848,Z 976.748,A 0.000,B 0.000,C 90.000,E1 350.735} C_DIS
LIN {X 0.167,Y -559.627,Z 976.745,A 0.000,B 0.000,C 90.000,E1 350.151} C_DIS
LIN {X 0.216,Y -565.070,Z 976.742,A 0.000,B 0.000,C 90.000,E1 349.454} C_DIS
LIN {X -0.247,Y -570.083,Z 976.738,A 0.000,B 0.000,C 90.000,E1 348.814} C_DIS
LIN {X -0.193,Y -572.923,Z 976.735,A 0.000,B 0.000,C 90.000,E1 348.398} C_DIS
LIN {X -0.032,Y -577.177,Z 976.732,A 0.000,B 0.000,C 90.000,E1 347.701} C_DIS
